// TIA Portal project "Centris" (V16)

(* hardware
DEVICE "S7-1200 station_1"  S7-1200 Station
   slot 0: "Rack_0"  S7-1200 Rack  Rack  V1.0
   slot 1: "PLC_1"  CPU 1214C DC/DC/Rly  6ES7 214-1HG40-0XB0  V4.4
*)

// ===== PLC "PLC_1"  CPU 1214C DC/DC/Rly =====

TYPE "UR__T2O_Robot"
   STRUCT
      "Controller major version" : USInt;
      "Controller minor version" : USInt;
      Reserved : UInt;
      "Robot mode" : USInt;
      "Real time machine seconds" : USInt;
      "Real time machine milliseconds" : UInt;
      "Real time machine minutes" : USInt;
      "Real time machine hours" : USInt;
      "Real time machine days" : UInt;
      "Robot current [A]" : Real;
      "PW: Is power on" : Bool;
      "PR: Is program running" : Bool;
      "TB: Is teach button pressed" : Bool;
      "PB: Is power button pressed" : Bool;
      Reserved_4 : Bool;
      Reserved_5 : Bool;
      Reserved_6 : Bool;
      Reserved_7 : Bool;
      Reserved_8_15 : USInt;
      Reserved_16_31 : UInt;
      "Speed slider fraction" : Real;
   END_STRUCT;
END_TYPE

TYPE "UR__T2O_Safety"
   STRUCT
      "Safety mode" : USInt;
      Reserved_1 : USInt;
      Reserved_2 : UInt;
      "NO: Is normal mode" : Bool;
      "RD: Is reduced mode" : Bool;
      "PS: Is protective stopped" : Bool;
      "RC: Is recovery mode" : Bool;
      "SS: Is safeguard stopped" : Bool;
      "SES: Is system emergency stopped" : Bool;
      "RES: Is robot emergency stopped" : Bool;
      "ES: Is emergency stopped" : Bool;
      "VL: Is violation" : Bool;
      "FT: Is fault" : Bool;
      "ST: Is stopped due to safety" : Bool;
      Reserved_11 : Bool;
      Reserved_12 : Bool;
      Reserved_13 : Bool;
      Reserved_14 : Bool;
      Reserved_15 : Bool;
      Reserved_16_31 : UInt;
   END_STRUCT;
END_TYPE

TYPE "UR__T2O_IOs"
   STRUCT
      "Standard digital inputs" : USInt;
      "Configurable digital inputs" : USInt;
      "Standard digital outputs" : USInt;
      "Configurable digital outputs" : USInt;
      "Analog I/O types" : USInt;
      Reserved_8_15 : USInt;
      Reserved_16_31 : UInt;
      "Standard analog input [A or V]" : Array[0..1] of Real;
      "Standard analog output [A or V]" : Array[0..1] of Real;
      "I/O current [A]" : Real;
      "Euromap67 input bits" : Array[0..31] of Bool;
      "Euromap67 output bits" : Array[0..31] of Bool;
      "Euromap67 24V voltage" : Real;
      "Euromap67 24V current" : Real;
   END_STRUCT;
END_TYPE

TYPE "UR__T2O_Tool"
   STRUCT
      "Tool mode" : USInt;
      Reserved_7_15 : USInt;
      Reserved_16_31 : UInt;
      "TDI: Tool Digital Inputs" : USInt;
      "TDO: Tool Digital Outputs" : USInt;
      "TAIT: Tool Analog Input Types" : USInt;
      Reserved_24_31 : USInt;
      "Tool analog input [A or V]" : Array[0..1] of Real;
      "Tool output voltage [V]" : Real;
      "Tool current [A]" : Real;
   END_STRUCT;
END_TYPE

TYPE "UR__O2T_floats"
   STRUCT
      Register : Array[0..11] of Real;
   END_STRUCT;
END_TYPE

TYPE "UR__O2T_ints"
   STRUCT
      Register : Array[0..11] of DInt;
   END_STRUCT;
END_TYPE

TYPE "UR__O2T_bits"
   STRUCT
      Register : Array[0..31] of Bool;
   END_STRUCT;
END_TYPE

TYPE "UR__O2T_Robot"
   STRUCT
      "SSM: Speed slider fraction mask" : Bool;
      Reserved_1 : Bool;
      Reserved_2 : Bool;
      Reserved_3 : Bool;
      Reserved_4 : Bool;
      Reserved_5 : Bool;
      Reserved_6 : Bool;
      Reserved_7 : Bool;
      Reserved_8_15 : USInt;
      Reserved_16_31 : UInt;
      "Speed slider fraction" : Real;
   END_STRUCT;
END_TYPE

TYPE "UR__O2T_IOs"
   STRUCT
      "Standard digital output mask" : USInt;
      "Configurable digital output mask" : USInt;
      "Standard digital outputs" : USInt;
      "Configurable digital outputs" : USInt;
      "AOM: Analog output mask" : USInt;
      "AOT: Analog output types" : USInt;
      "TDOM: Tool digital output mask" : USInt;
      "TDO: Tool digital output" : USInt;
      "Standard analog output" : Array[0..1] of Real;
   END_STRUCT;
END_TYPE

TYPE "Recipe_Data"
   STRUCT
      ID : DInt;   // ID
      ServoSpeed : DInt;
      ServoForceRamp : DInt;
      ServoForce : DInt;
      ServoRedPos : DInt;
      ServoBluePos : DInt;
      ServoYellowPos : DInt;
      "IV RedProgram" : Int;
      "IV BlueProgram" : Int;
      "IV YellowProgram" : Int;
   END_STRUCT;
END_TYPE

TYPE "Latch"
   STRUCT
      Latch : Bool;
      Ons : Bool;
      Action : Bool;
      Delay : Bool;
      PB : Bool;
      TON : IEC_TIMER;
   END_STRUCT;
END_TYPE

TYPE "UR_9_O2T_Registers"
   STRUCT
      Bits : "UR__O2T_bits";
      Ints : "UR__O2T_ints";
      Floats : "UR__O2T_floats";
   END_STRUCT;
END_TYPE

TYPE "UR_8_O2T_Robot_IO"
   STRUCT
      Robot : "UR__O2T_Robot";
      IOs : "UR__O2T_IOs";
   END_STRUCT;
END_TYPE

TYPE "UR_7_T2O_FloatRegisters"
   STRUCT
      Register : Array[0..23] of Real;
   END_STRUCT;
END_TYPE

TYPE "UR_6_T2O_IntRegisters"
   STRUCT
      Register : Array[0..23] of DInt;
   END_STRUCT;
END_TYPE

TYPE "UR_5_T2O_BitRegisters"
   STRUCT
      Register : Array[0..63] of Bool;
   END_STRUCT;
END_TYPE

TYPE "UR_4_T2O_TCP"
   STRUCT
      "TCP Position (X,Y,Z) [m]" : Array[0..2] of Real;
      "TCP Position (RX,RY,RZ) [rad]" : Array[0..2] of Real;
      "TCP velocity (X,Y,Z) [m/s]" : Array[0..2] of Real;
      "TCP velocity (RX,RY,RZ) [rad/s]" : Array[0..2] of Real;
      "TCP force (X,Y,Z) [N]" : Array[0..2] of Real;
      "TCP torque (X,Y,Z) [Nm]" : Array[0..2] of Real;
      "TCP force scalar [N]" : Real;
   END_STRUCT;
END_TYPE

TYPE "UR_3_T2O_Joints"
   STRUCT
      "Joint position [rad]" : Array[0..5] of Real;
      "Joint velocity [rad/s]" : Array[0..5] of Real;
      "Joint current [A]" : Array[0..5] of Real;
      "Joint temperature [°C]" : Array[0..5] of Real;
      "Joint mode" : Array[0..5] of USInt;
      Reserved_9 : UInt;
   END_STRUCT;
END_TYPE

TYPE "UR_2_T2O_IO"
   STRUCT
      IOs : "UR__T2O_IOs";
      Tool : "UR__T2O_Tool";
   END_STRUCT;
END_TYPE

TYPE "UR_1_T2O_State"
   STRUCT
      Robot : "UR__T2O_Robot";
      Safety : "UR__T2O_Safety";
   END_STRUCT;
END_TYPE

TYPE "Festo Control IN/OUT"
   STRUCT
      "Enable Connection" : Bool;
      "Device Type" : String;
      "Enable FPC" : Bool;
      "Enable FHPPPlus_In" : Int;
      "Enable FHPPPlus_Out" : Int;
      "IP_Oct#1" : Int;
      "IP_Oct#2" : Int;
      "IP_Oct#3" : Int;
      "IP_Oct#4" : Int;
      "Interface ID" : Hw_Any;
      "Connection ID" : Int;
      TimeOut : Time;
      "Com Enabled" : Bool;
      Error : Bool;
      Status : "DT_FML_STATUS";
      "Enable Control" : Bool;
      "Stop Control" : Bool;
      "Halt Control" : Bool;
      "Brake Control" : Bool;
      "Reset Control" : Bool;
      "HMI Access" : Bool;
      "Operation Mode" : Int;
      "Start Task" : Bool;
      "Start Homing" : Bool;
      "Jog Positive" : Bool;
      "Jog Negative" : Bool;
      "Teach Value" : Bool;
      "Clear Rem Position" : Bool;
      Relative : Bool;
      "Desactivate Stroke Limit" : Bool;
      "Execute Function" : Bool;
      "Record Number" : Int;
      "Set Function Number" : Int;
      "Set Function Group" : Int;
      "Set Velocity" : DInt;
      "Set Position Pre" : DInt;
      "Set Position Val" : DInt;
      "Set Force Ramp" : DInt;
      "Set Force" : DInt;
      "Set Rot Ramp" : DInt;
      "Set Rot Speed" : DInt;
      "Spare 1" : DInt;
      "Drive Enabled" : Bool;
      "Driver Ready" : Bool;
      Warning : Bool;
      "Driver Faulted" : Bool;
      "Driver Supply Voltage Present" : Bool;
      "Control FCT_HMI" : Bool;
      "Actual Operation Mode" : Int;
      "Halt Not Active" : Bool;
      "Start ACK" : Bool;
      "PLC Master Control" : Bool;
      "Teach ACK" : Bool;
      "Drive Moving" : Bool;
      "Drag Error" : Bool;
      "Stand Still Control" : Bool;
      "Homing Valid" : Bool;
      "Actual Record Number" : Int;
      RC1 : Bool;
      RCC : Bool;
      "Velocity Limit Reached" : Bool;
      "Stroke Limit Reached" : Bool;
      "Function Is Active" : Bool;
      "Actual Function Number" : Int;
      "Actual Function Group" : Int;
      "Actual Position" : DInt;
      "Actual Velocity" : DInt;
      "Actual Force" : DInt;
      "Actual Rot Ramp" : DInt;
      "Actual Rot Speed" : DInt;
      WatchDog_Timer_ON : Time;
      WatchDog_Timer_OFF : Time;
      WatrchDog_Reset : Bool;
      "Execute PNU" : Bool;
      Write : Bool;
      DatatypeWR : Int;
      PNU : Int;
      Subindex : Int;
      Value : DInt;
      Done : Bool;
      ErrorPNU : Bool;
      ActPNU : Int;
      ActSubindex : Int;
      ActValue : DInt;
      DatatypeRD : Int;
      StatusPNU : "DT_FML_STATUS";
      WatchDog_Timer : Array[0..10] of IEC_TIMER;
      WatchDog_Reset_Connection : Bool;
      WatchDog_Reset_Device : Bool;
      WatchDog_Reset_Control : Bool;
      "PNU BOOL" : Bool;
      "Manual Buffer" : DInt;
      "Position Buffer" : DInt;
      Delay : Array[0..10] of IEC_TIMER;
      SetProgram_Red : Int;
      SetProgram_Blue : Int;
      SetProgram_Yellow : Int;
      Set_Red_Position : DInt;
      Set_Blue_Position : DInt;
      Set_Yellow_Position : DInt;
      Red_StartTask : Bool;
      Blue_StartTask : Bool;
      Yellow_StartTask : Bool;
      Home_StartTask : Bool;
      RedPos : Bool;
      BluePos : Bool;
      YellowPos : Bool;
      HomePos : Bool;
      Available_StartTask : Bool;
   END_STRUCT;
END_TYPE

TYPE "Safety"
   STRUCT
      "EStops OK" : Bool;
      "Safety Guards OK" : Bool;
      "Interlocks OK" : Bool;
      "SSD Robots OK" : Bool;
      "SSD Servos OK" : Bool;
      "Safety Doors OK" : Bool;
      "Safety Relays OK" : Bool;
      "SSD vfd Motors OK" : Bool;
      "Safety Curtains OK" : Bool;
      "Safety Devices OK" : Bool;
      "Communication Devices OK" : Bool;
      "Clear Error Devices OK" : Bool;
      "Clear Fault Devices OK" : Bool;
      "Safety Air OK" : Bool;
      "Power ON Start" : Bool;
      "Enable System Start" : Bool;
      "All Safety Devices OK" : Bool;
   END_STRUCT;
END_TYPE

TYPE "Mode"
   STRUCT
      "Run Stop" : Bool;
      "Run Auto" : Bool;
      "Run Start" : Bool;
      "Run Manual" : Bool;
      "Run Dry Cycle" : Bool;
      "Enable Cycle Stop" : Bool;
      "Enable Auto" : Bool;
      "Enable Start" : Bool;
      "Enable Manual" : Bool;
      "Enable Dry Cycle" : Bool;
      "Enable Home" : Bool;
      "Run Home" : Bool;
   END_STRUCT;
END_TYPE

TYPE "Push_Buttons"
   STRUCT
      AllHome : Bool;
      Stop : Bool;
      Auto : Bool;
      Start : Bool;
      StartProcess : Bool;
      Manual : Bool;
      DryCycle : Bool;
      Reset : Bool;
      Trigger : Bool;
      IVProgramRed : Bool;
      IVProgramBLue : Bool;
      IVProgramYellow : Bool;
      FestoRedPos : Bool;
      FestoBluePos : Bool;
      FestoYellowPos : Bool;
      FestoHomePos : Bool;
      "UR RedPos" : Bool;
      "UR BluePos" : Bool;
      "UR YellowPos" : Bool;
      "UR HomePos" : Bool;
      RecipeSelect : Array[0..5] of Bool;
      RecipeEdit : Array[0..5] of Bool;
      Saving : Bool;
      ResetBuffer : Bool;
      AutoPlay : Bool;
      AutoInit : Bool;
      StartProgram : Bool;
      StopProgram : Bool;
      PauseProgram : Bool;
      FreeDrive : Bool;
      FestoReset : Bool;
      URReset : Bool;
      MainReset : Bool;
      VisionReset : Bool;
      FaultsReset : Bool;
      WarningsReset : Bool;
   END_STRUCT;
END_TYPE

TYPE "UR_O2T"
   STRUCT
      "Robot IO" : "UR_8_O2T_Robot_IO";
      "Reg 1" : "UR_9_O2T_Registers";
      "Reg 2" : "UR_9_O2T_Registers";
   END_STRUCT;
END_TYPE

TYPE "Alarms"
   STRUCT
      Fault : Array[0..100] of Bool;
      Warning : Array[0..100] of Bool;
      Status : Array[0..100] of Bool;
      Clear : Array[0..100] of Bool;
      ClearFaults : Bool;
      ClearWarnings : Bool;
      ClearStatus : Bool;
      Fton : Array[0..100] of IEC_TIMER;
      Wton : Array[0..100] of IEC_TIMER;
      Ston : Array[0..100] of IEC_TIMER;
   END_STRUCT;
END_TYPE

TYPE "Ctlr_Recipe"
   STRUCT
      "Actual Running Recipe" : "Recipe_Data";
      "Editing Recipe" : "Recipe_Data";
      "Selected Recipe" : "Recipe_Data";
      Saving : "Latch";
      Select : "Latch";
      Edit : "Latch";
      MoveBit : Array[0..5] of Bool;
      EditBit : Array[0..5] of Bool;
      "Any Recipe Selected" : Bool;
      "None Recipe Selected" : Bool;
      "End Of Sequence" : Bool;
      "Cycle Running" : Bool;
   END_STRUCT;
END_TYPE

TYPE "iv_500ca_in"
   STRUCT
      "Trigger response" : Bool;   // Command Status Bits Address 0:0
      "Master registration response" : Bool;   // Command Status Bits Address 0:1
      "Program switching response" : Bool;   // Command Status Bits Address 0:2
      "Warning clear response" : Bool;   // Command Status Bits Address 0:3
      "Statistics reset response" : Bool;   // Command Status Bits Address 0:4
      "Buffer clear response" : Bool;   // Command Status Bits Address 0:5
      "Command Status Bits Address 0:6" : Bool;   // Command Status Bits Address 0:6
      "Command Status Bits Address 0:7" : Bool;   // Command Status Bits Address 0:7
      "Trigger failed" : Bool;   // Command Status Bits Address 1:0
      "Master registration failed" : Bool;   // Command Status Bits Address 1:1
      "Program switching failed" : Bool;   // Command Status Bits Address 1:2
      "Command Status Bits Address 1:3" : Bool;   // Command Status Bits Address 1:3
      "Command Status Bits Address 1:4" : Bool;   // Command Status Bits Address 1:4
      "Command Status Bits Address 1:5" : Bool;   // Command Status Bits Address 1:5
      "Command Status Bits Address 1:6" : Bool;   // Command Status Bits Address 1:6
      "Command Status Bits Address 1:7" : Bool;   // Command Status Bits Address 1:7
      "Result available" : Bool;   // Command Status Bits Address 2:0
      "Result update complete" : Bool;   // Command Status Bits Address 2:1
      Busy : Bool;   // Command Status Bits Address 2:2
      Imaging : Bool;   // Command Status Bits Address 2:3
      RUN : Bool;   // Command Status Bits Address 2:4
      Ready : Bool;   // Command Status Bits Address 2:5
      "Command Status Bits Address 2:6" : Bool;   // Command Status Bits Address 2:6
      "Command Status Bits Address 2:7" : Bool;   // Command Status Bits Address 2:7
      "Command Status Bits Address 3:0" : Bool;   // Command Status Bits Address 3:0
      "Command Status Bits Address 3:1" : Bool;   // Command Status Bits Address 3:1
      "Command Status Bits Address 3:2" : Bool;   // Command Status Bits Address 3:2
      "Command Status Bits Address 3:3" : Bool;   // Command Status Bits Address 3:3
      "Command Status Bits Address 3:4" : Bool;   // Command Status Bits Address 3:4
      "Buffer overrun status" : Bool;   // Command Status Bits Address 3:5
      "Warning status" : Bool;   // Command Status Bits Address 3:6
      "Error status" : Bool;   // Command Status Bits Address 3:7
      "Overall judgment" : Bool;   // Device Results Bits Address 0:0
      "Position correction" : Bool;   // Device Results Bits Address 0:1
      "Logic 1" : Bool;   // Device Results Bits Address 0:2
      "Logic 2" : Bool;   // Device Results Bits Address 0:3
      "Logic 3" : Bool;   // Device Results Bits Address 0:4
      "Logic 4" : Bool;   // Device Results Bits Address 0:5
      "Overall judgement NG" : Bool;   // Device Results Bits Address 0:6
      "Device Results Bits Address 0:7" : Bool;   // Device Results Bits Address 0:7
      "Device Results Bits Address 1:0" : Bool;   // Device Results Bits Address 1:0
      "Device Results Bits Address 1:1" : Bool;   // Device Results Bits Address 1:1
      "Device Results Bits Address 1:2" : Bool;   // Device Results Bits Address 1:2
      "Device Results Bits Address 1:3" : Bool;   // Device Results Bits Address 1:3
      "Device Results Bits Address 1:4" : Bool;   // Device Results Bits Address 1:4
      "Device Results Bits Address 1:5" : Bool;   // Device Results Bits Address 1:5
      "Device Results Bits Address 1:6" : Bool;   // Device Results Bits Address 1:6
      "Device Results Bits Address 1:7" : Bool;   // Device Results Bits Address 1:7
      "Tool 1" : Bool;   // Device Results Bits Address 2:0
      "Tool 2" : Bool;   // Device Results Bits Address 2:1
      "Tool 3" : Bool;   // Device Results Bits Address 2:2
      "Tool 4" : Bool;   // Device Results Bits Address 2:3
      "Tool 5" : Bool;   // Device Results Bits Address 2:4
      "Tool 6" : Bool;   // Device Results Bits Address 2:5
      "Tool 7" : Bool;   // Device Results Bits Address 2:6
      "Tool 8" : Bool;   // Device Results Bits Address 2:7
      "Tool 9" : Bool;   // Device Results Bits Address 3:0
      "Tool 10" : Bool;   // Device Results Bits Address 3:1
      "Tool 11" : Bool;   // Device Results Bits Address 3:2
      "Tool 12" : Bool;   // Device Results Bits Address 3:3
      "Tool 13" : Bool;   // Device Results Bits Address 3:4
      "Tool 14" : Bool;   // Device Results Bits Address 3:5
      "Tool 15" : Bool;   // Device Results Bits Address 3:6
      "Tool 16" : Bool;   // Device Results Bits Address 3:7
      "Error code" : Word;   // Device Status Words Address 0 to 1
      "Warning code" : Word;   // Device Status Words Address 2 to 3
      "Number of remaining buffers" : Word;   // Device Status Words Address 4 to 5
      Checksum : Word;   // Device Status Words Address 6 to 7
      "Current program No." : Word;   // Device Status Words Address 8 to 9
      "Program No. during judgment" : Word;   // Device Status Words Address 10 to 11
      "Result No." : Word;   // Device Status Words Address 12 to 13
      "Processing time" : Word;   // Device Status Words Address 14 to 15
      "Processing time Max" : Word;   // Device Statistics Address 0 to 1
      "Processing time Min" : Word;   // Device Statistics Address 2 to 3
      "Processing time Ave" : Word;   // Device Statistics Address 4 to 5
      "Device Statistics Address 6 to 7" : Word;   // Device Statistics Address 6 to 7
      "Number of triggers" : DWord;   // Device Statistics Address 8 to 11
      "Number of OKs" : DWord;   // Device Statistics Address 12 to 15
      "Number of NGs" : DWord;   // Device Statistics Address 16 to 19
      "Number of trigger errors" : DWord;   // Device Statistics Address 20 to 23
      "Device Statistics Address 24 to 27" : DWord;   // Device Statistics Address 24 to 27
      "Position correction tool matching rate" : Word;   // Position Adjust Result Address 0 to 1
      "Position correction score MAX" : Word;   // Position Adjust Result Address 2 to 3
      "Position correction score MIN" : Word;   // Position Adjust Result Address 4 to 5
      "Position correction tool Threshold value" : Word;   // Position Adjust Result Address 6 to 7
      "Position Adjust Result Address 8 to 9" : Word;   // Position Adjust Result Address 8 to 9
      "Position Adjust Result Address 10 to 11" : Word;   // Position Adjust Result Address 10 to 11
      "Position Adjust Result Address 12 to 13" : Word;   // Position Adjust Result Address 12 to 13
      "Position Adjust Result Address 14 to 15" : Word;   // Position Adjust Result Address 14 to 15
      "Position Adjust Result Address 16 to 17" : Word;   // Position Adjust Result Address 16 to 17
      "Position Adjust Result Address 18 to 19" : Word;   // Position Adjust Result Address 18 to 19
      "Tool 1 matching rate" : Word;   // Tool Result Address 0 to 1
      "Tool 1 matching rate MAX" : Word;   // Tool Result Address 2 to 3
      "Tool 1 matching rate MIN" : Word;   // Tool Result Address 4 to 5
      "Tool 1 lower limit value" : Word;   // Tool Result Address 6 to 7
      "Tool 1 upper limit value" : Word;   // Tool Result Address 8 to 9
      "Tool Result Address 10" : Byte;   // Tool Result Address 10
      "Tool Result Address 11" : Byte;   // Tool Result Address 11
      "Tool Result Address 12" : Byte;   // Tool Result Address 12
      "Tool Result Address 13" : Byte;   // Tool Result Address 13
      "Tool Result Address 14" : Byte;   // Tool Result Address 14
      "Tool Result Address 15" : Byte;   // Tool Result Address 15
      "Tool Result Address 16" : Byte;   // Tool Result Address 16
      "Tool Result Address 17" : Byte;   // Tool Result Address 17
      "Tool Result Address 18" : Byte;   // Tool Result Address 18
      "Tool Result Address 19" : Byte;   // Tool Result Address 19
   END_STRUCT;
END_TYPE

TYPE "iv_500ca_out"
   STRUCT
      "Trigger request" : Bool;   // Command Control 1:0
      "Master registration request" : Bool;   // Command Control 1:1
      "Programm switching request" : Bool;   // Command Control 1:2
      "Warning clear request" : Bool;   // Command Control 1:3
      "Statistics reset request" : Bool;   // Command Control 1:4
      "Buffer clear request" : Bool;   // Command Control 1:5
      "Command Control 1:6" : Bool;   // Command Control 1:6
      "Command Control 1:7" : Bool;   // Command Control 1:7
      "Result acquisition complete notification" : Bool;   // Command Control 2:0
      "Command Control 2:1" : Bool;   // Command Control 2:1
      "Command Control 2:2" : Bool;   // Command Control 2:2
      "Command Control 2:3" : Bool;   // Command Control 2:3
      "Command Control 2:4" : Bool;   // Command Control 2:4
      "Command Control 2:5" : Bool;   // Command Control 2:5
      "Command Control 2:6" : Bool;   // Command Control 2:6
      "Command Control 2:7" : Bool;   // Command Control 2:7
      "Command Control 3" : Byte;   // Command Control 3
      "Programm No." : Word;   // Command Control 4 to 5
      "Command Control 6" : Byte;   // Command Control 6
      "Command Control 7" : Byte;   // Command Control 7
      "Command Control 8" : Byte;   // Command Control 8
      "Command Control 9" : Byte;   // Command Control 9
      "Command Control 10" : Byte;   // Command Control 10
      "Command Control 11" : Byte;   // Command Control 11
   END_STRUCT;
END_TYPE

TYPE "IV_Ctrl"
   STRUCT
      CommActive : Bool;
      ResetBuffer : Bool;
      InspectionComplete : Bool;
      InspectionOK : Bool;
      InspectionNOK : Bool;
      InspectionRequest : Bool;
      InspectReqTimeout : IEC_TIMER;
      ConnectionFault : Bool;
      CameraFault : Bool;
      InspectionRequestTimeoutFault : Bool;
      "Clear Results" : Bool;
      Trigger : Bool;
      OKRed : Bool;
      NOKRed : Bool;
      OKBlue : Bool;
      NOKBlue : Bool;
      OKYellow : Bool;
      NOKYellow : Bool;
      AllClearResults : Bool;
      NOKAllResults : Bool;
      "Run Red" : Bool;
      "Run Blue" : Bool;
      "Run Yellow" : Bool;
      OKAnyResult : Bool;
   END_STRUCT;
END_TYPE

TYPE "PLC_Digital_IN"
   STRUCT
      START : Bool;
      RESET : Bool;
      ESTOP : Bool;
      "I0.3" : Bool;
      "I0.4" : Bool;
      "I0.5" : Bool;
      "I0.6" : Bool;
      "I0.7" : Bool;
      "I1.0" : Bool;
      "I1.1" : Bool;
      "I1.2" : Bool;
      "I1.3" : Bool;
      "I1.4" : Bool;
      "I1.5" : Bool;
      "I1.6" : Bool;
      "I1.7" : Bool;
   END_STRUCT;
END_TYPE

TYPE "PLC_Digital_Out"
   STRUCT
      "Q0.0" : Bool;
      "Q0.1" : Bool;
      "Q0.2" : Bool;
      "Q0.3" : Bool;
      "Q0.4" : Bool;
      "Q0.5" : Bool;
      "Q0.6" : Bool;
      "Q0.7" : Bool;
      "Q1.0" : Bool;
      "Q1.1" : Bool;
      "Q1.2" : Bool;
      "Q1.3" : Bool;
      "Q1.4" : Bool;
      "Q1.5" : Bool;
      "Q1.6" : Bool;
      "Q1.7" : Bool;
   END_STRUCT;
END_TYPE

TYPE "UR_T2O"
   STRUCT
      State : "UR_1_T2O_State";
      IO : "UR_2_T2O_IO";
      Joints : "UR_3_T2O_Joints";
      TCP : "UR_4_T2O_TCP";
      Bits : "UR_5_T2O_BitRegisters";
      Ints : "UR_6_T2O_IntRegisters";
      Floats : "UR_7_T2O_FloatRegisters";
   END_STRUCT;
END_TYPE

TYPE "Production"
   STRUCT
      Ton : Array[0..12] of IEC_TIMER;
      Seq : Array[0..12] of Bool;
      Permissive : Array[0..12] of Bool;
      Clear : Array[0..12] of Bool;
      "Clear Sequence" : Bool;
      "All Home OK" : Bool;
      ReplaceIN : Array[0..15] of Bool;
      "Cycle ResetAllMemories" : Bool;
      "UR Home OK" : Bool;
      "UR Program" : DInt;
      "UR EndRoutine" : Bool;
      "All Memories StatusClear" : Bool;
      StatusSeq : Bool;
      StatusStart : Bool;
      StatusHome : Bool;
      "UR RunRed" : Bool;
      "UR RunBlue" : Bool;
      "UR RunYellow" : Bool;
      "UR Start Program" : Bool;
   END_STRUCT;
END_TYPE

// folder: FML DATATYPES

TYPE "DT_FML_STATUS"
   STRUCT
      Err : Bool;
      Cat : Int;
      ID : DInt;
   END_STRUCT;
END_TYPE

TYPE "DT_FML_PRM_FILE"
   STRUCT
      Control : Int;
      BitSequenceNr : Int;
      Data : Array[1..6] of Byte;
   END_STRUCT;
END_TYPE

TYPE "DT_FML_REF"
   STRUCT
      InData : Struct
         FHPP : Array[1..16] of Byte;
         FPC : Array[1..8] of Byte;
         FHPPplus : Array[1..10] of DInt;
      END_STRUCT;
      OutData : Struct
         FHPP : Array[1..16] of Byte;
         FPC : Array[1..8] of Byte;
         FHPPplus : Array[1..10] of DInt;
      END_STRUCT;
      Modbus : Bool;
      DeviceType : String[16];
      MemberID : Int;
      MemberIDmax : Int;
      Done : Bool;
      Err : Bool;
      PNU : Word;
      ActPNU : Word;
      ReqID : Int;
      RespID : Int;
      FPCC_Modus : Byte;
      FPCS_Modus : Byte;
      FPCC_Packet : "DT_FML_PRM_FILE";
      FPCS_Packet : "DT_FML_PRM_FILE";
      Subindex : Byte;
      ActSubindex : Byte;
      DatatypeWR : Byte;
      DatatypeRD : Byte;
      ParamValueWR : DInt;
      ParamValueRD : DInt;
   END_STRUCT;
END_TYPE

TYPE "DT_MB_CLIENT_INPUT"
   STRUCT
      REQ : Bool;
      DISCONNECT : Bool;
      Done : Bool;
      Busy : Bool;
      Error : Bool;
      MB_MODE : USInt;
      MB_DATA_ADDR : UDInt;
      MB_DATA_LEN : UInt;
   END_STRUCT;
END_TYPE

TYPE "DT_FML_PRM_DESCRIPTION"
   STRUCT
      PNU : Word;
      SUBINDEX : Byte;
      ACCESS : Byte;
      VALUE : DInt;
      LENGTH : Byte;
   END_STRUCT;
END_TYPE

TYPE "DT_FML_PRM_DIAGMESSAGE"
   STRUCT
      Event : DInt;
      MsgNumber : DInt;
      TimeStamp : DWord;
   END_STRUCT;
END_TYPE

// folder: (top level)

DATA_BLOCK "DB"   // DB1
{ S7_Optimized_Access := 'FALSE' }
VERSION : 0.1
   VAR
      Alarm : "Alarms";
      Prod : "Production";
      UR : "Production";
      Ctrl_Recipe : "Ctlr_Recipe";
      FESTO : "Festo Control IN/OUT";
      AUTO : "Festo Control IN/OUT";
      MANUAL : "Festo Control IN/OUT";
      OP : "Festo Control IN/OUT";
      HMI : "Push_Buttons";
      "Mod" : "Mode";
      Safe : "Safety";
      "IV Ctrl" : "IV_Ctrl";
      I : "PLC_Digital_IN";
      "N/A" : Bool;
   END_VAR
BEGIN
END_DATA_BLOCK

DATA_BLOCK "FHPP_MB_CLIENT_DB"   // DB7
{ S7_Optimized_Access := 'TRUE' }
AUTHOR : FESTO
FAMILY : E-DRIVE
VERSION : 5.1
// stored: InstanceOfName FHPP_MB_CLIENT
"FHPP_MB_CLIENT"
BEGIN
END_DATA_BLOCK

DATA_BLOCK "FHPP_CTRL_DB"   // DB8
{ S7_Optimized_Access := 'TRUE' }
AUTHOR : FESTO
FAMILY : E-DRIVE
VERSION : 5.1
// stored: InstanceOfName FHPP_CTRL
"FHPP_CTRL"
BEGIN
END_DATA_BLOCK

DATA_BLOCK "FPC_PNU_DB"   // DB9
{ S7_Optimized_Access := 'TRUE' }
AUTHOR : FESTO
FAMILY : E-DRIVE
VERSION : 5.1
// stored: InstanceOfName FPC_PNU
"FPC_PNU"
BEGIN
END_DATA_BLOCK

// folder: RECIPE

DATA_BLOCK "Recipe"   // DB2
{ S7_Optimized_Access := 'TRUE' }
VERSION : 0.1
BEGIN
END_DATA_BLOCK

// folder: UTILITIES OR DEVICES/FESTO

DATA_BLOCK "Global_Modbuss_CMMO"   // DB6
{ S7_Optimized_Access := 'TRUE' }
VERSION : 0.1
   VAR
      CMMO_REF : "DT_FML_REF";
   END_VAR
BEGIN
END_DATA_BLOCK

DATA_BLOCK "gBUFFER_MODBUS"   // DB100
TITLE = Buffer for MB_Client
{ S7_Optimized_Access := 'FALSE' }
AUTHOR : FESTO
FAMILY : E-Drives
VERSION : 4.1
   VAR
      ModbusBuffer : Array[1..100] of Byte;
   END_VAR
BEGIN
END_DATA_BLOCK

// folder: UTILITIES OR DEVICES/MODBUS TCP LABVIEW

DATA_BLOCK "Labview"   // DB3
{ S7_Optimized_Access := 'FALSE' }
VERSION : 0.1
BEGIN
END_DATA_BLOCK

DATA_BLOCK "MBConfig"   // DB4
{ S7_Optimized_Access := 'FALSE' }
VERSION : 0.1
BEGIN
END_DATA_BLOCK

DATA_BLOCK "MBData"   // DB5
{ S7_Optimized_Access := 'FALSE' }
VERSION : 0.1
BEGIN
END_DATA_BLOCK

// folder: (top level)

ORGANIZATION_BLOCK "Main"   // OB1, LAD, ProgramCycle
TITLE = "Main Program Sweep (Cycle)"
{ S7_Optimized_Access := 'TRUE' }
VERSION : 0.1
   VAR_INPUT
      Initial_Call : Bool;   // Initial call of this OB
      Remanence : Bool;   // =True, if remanent data are available
   END_VAR
BEGIN

REGION Network 1: CALL_LADDER
END_REGION

REGION Network 2: FESTO MODBUS CLIENT
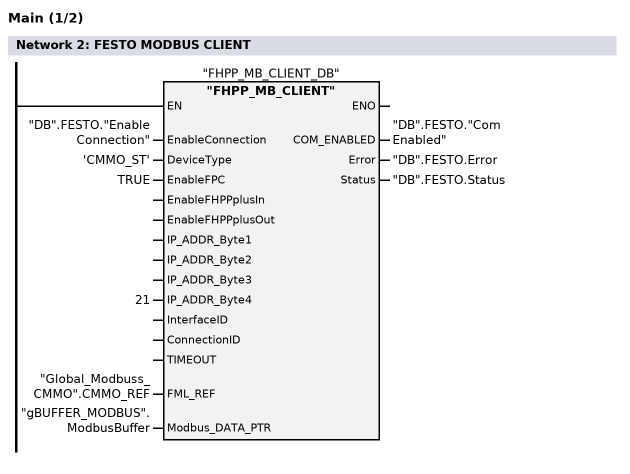
   RUNG wire#powerrail
      "FHPP_MB_CLIENT_DB"(EnableConnection := "DB".FESTO."Enable Connection", DeviceType := 'CMMO_ST', EnableFPC := TRUE, EnableFHPPplusIn :=, EnableFHPPplusOut :=, IP_ADDR_Byte1 :=, IP_ADDR_Byte2 :=, IP_ADDR_Byte3 :=, IP_ADDR_Byte4 := 21, InterfaceID :=, ConnectionID :=, TIMEOUT :=, FML_REF := "Global_Modbuss_CMMO".CMMO_REF, Modbus_DATA_PTR := "gBUFFER_MODBUS".ModbusBuffer, COM_ENABLED => "DB".FESTO."Com Enabled", Error => "DB".FESTO.Error, Status => "DB".FESTO.Status)
   END_RUNG
   // the same network as SCL:
   "FHPP_MB_CLIENT_DB"(EnableConnection := "DB".FESTO."Enable Connection",   // "FHPP_MB_CLIENT"
                       DeviceType := 'CMMO_ST',
                       EnableFPC := TRUE,
                       IP_ADDR_Byte4 := 21,
                       FML_REF := "Global_Modbuss_CMMO".CMMO_REF,
                       Modbus_DATA_PTR := "gBUFFER_MODBUS".ModbusBuffer,
                       COM_ENABLED => "DB".FESTO."Com Enabled",
                       Error => "DB".FESTO.Error,
                       Status => "DB".FESTO.Status);
END_REGION

REGION Network 3: FESTO DRIVER CONTROL
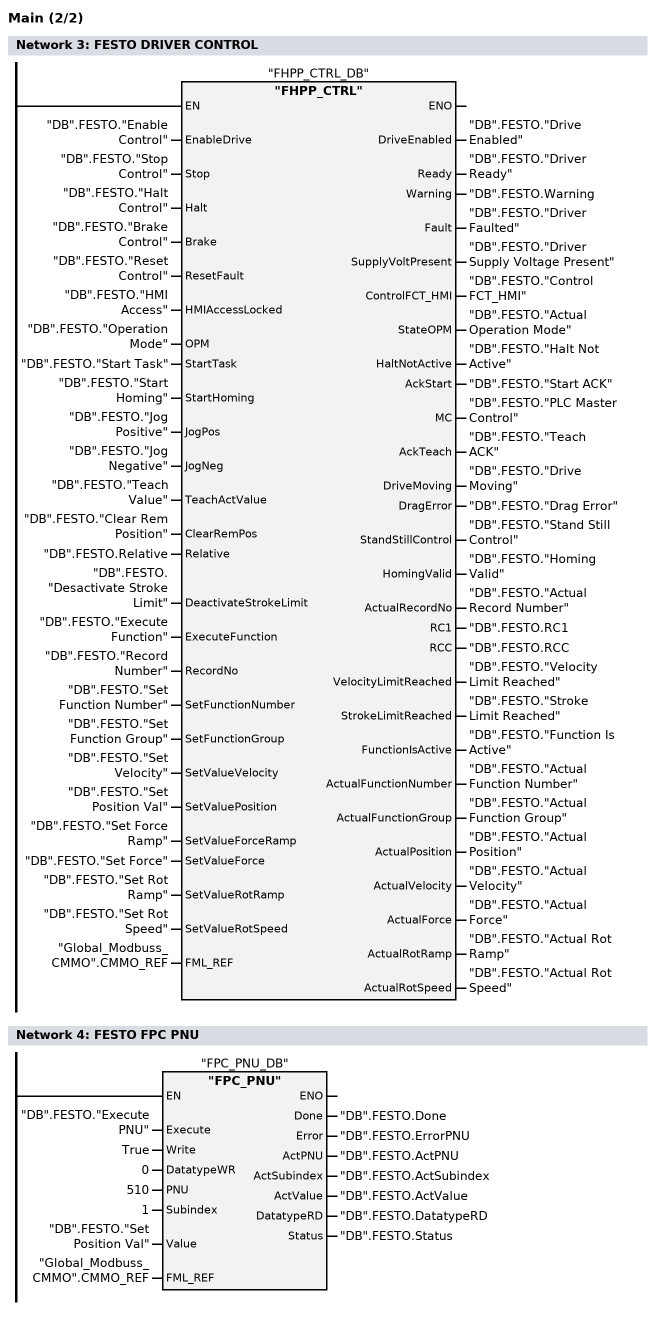
   RUNG wire#powerrail
      "FHPP_CTRL_DB"(EnableDrive := "DB".FESTO."Enable Control", Stop := "DB".FESTO."Stop Control", Halt := "DB".FESTO."Halt Control", Brake := "DB".FESTO."Brake Control", ResetFault := "DB".FESTO."Reset Control", HMIAccessLocked := "DB".FESTO."HMI Access", OPM := "DB".FESTO."Operation Mode", StartTask := "DB".FESTO."Start Task", StartHoming := "DB".FESTO."Start Homing", JogPos := "DB".FESTO."Jog Positive", JogNeg := "DB".FESTO."Jog Negative", TeachActValue := "DB".FESTO."Teach Value", ClearRemPos := "DB".FESTO."Clear Rem Position", Relative := "DB".FESTO.Relative, DeactivateStrokeLimit := "DB".FESTO."Desactivate Stroke Limit", ExecuteFunction := "DB".FESTO."Execute Function", RecordNo := "DB".FESTO."Record Number", SetFunctionNumber := "DB".FESTO."Set Function Number", SetFunctionGroup := "DB".FESTO."Set Function Group", SetValueVelocity := "DB".FESTO."Set Velocity", SetValuePosition := "DB".FESTO."Set Position Val", SetValueForceRamp := "DB".FESTO."Set Force Ramp", SetValueForce := "DB".FESTO."Set Force", SetValueRotRamp := "DB".FESTO."Set Rot Ramp", SetValueRotSpeed := "DB".FESTO."Set Rot Speed", FML_REF := "Global_Modbuss_CMMO".CMMO_REF, DriveEnabled => "DB".FESTO."Drive Enabled", Ready => "DB".FESTO."Driver Ready", Warning => "DB".FESTO.Warning, Fault => "DB".FESTO."Driver Faulted", SupplyVoltPresent => "DB".FESTO."Driver Supply Voltage Present", ControlFCT_HMI => "DB".FESTO."Control FCT_HMI", StateOPM => "DB".FESTO."Actual Operation Mode", HaltNotActive => "DB".FESTO."Halt Not Active", AckStart => "DB".FESTO."Start ACK", MC => "DB".FESTO."PLC Master Control", AckTeach => "DB".FESTO."Teach ACK", DriveMoving => "DB".FESTO."Drive Moving", DragError => "DB".FESTO."Drag Error", StandStillControl => "DB".FESTO."Stand Still Control", HomingValid => "DB".FESTO."Homing Valid", ActualRecordNo => "DB".FESTO."Actual Record Number", RC1 => "DB".FESTO.RC1, RCC => "DB".FESTO.RCC, VelocityLimitReached => "DB".FESTO."Velocity Limit Reached", StrokeLimitReached => "DB".FESTO."Stroke Limit Reached", FunctionIsActive => "DB".FESTO."Function Is Active", ActualFunctionNumber => "DB".FESTO."Actual Function Number", ActualFunctionGroup => "DB".FESTO."Actual Function Group", ActualPosition => "DB".FESTO."Actual Position", ActualVelocity => "DB".FESTO."Actual Velocity", ActualForce => "DB".FESTO."Actual Force", ActualRotRamp => "DB".FESTO."Actual Rot Ramp", ActualRotSpeed => "DB".FESTO."Actual Rot Speed")
   END_RUNG
   // the same network as SCL:
   "FHPP_CTRL_DB"(EnableDrive := "DB".FESTO."Enable Control",   // "FHPP_CTRL"
                  Stop := "DB".FESTO."Stop Control",
                  Halt := "DB".FESTO."Halt Control",
                  Brake := "DB".FESTO."Brake Control",
                  ResetFault := "DB".FESTO."Reset Control",
                  HMIAccessLocked := "DB".FESTO."HMI Access",
                  OPM := "DB".FESTO."Operation Mode",
                  StartTask := "DB".FESTO."Start Task",
                  StartHoming := "DB".FESTO."Start Homing",
                  JogPos := "DB".FESTO."Jog Positive",
                  JogNeg := "DB".FESTO."Jog Negative",
                  TeachActValue := "DB".FESTO."Teach Value",
                  ClearRemPos := "DB".FESTO."Clear Rem Position",
                  Relative := "DB".FESTO.Relative,
                  DeactivateStrokeLimit := "DB".FESTO."Desactivate Stroke Limit",
                  ExecuteFunction := "DB".FESTO."Execute Function",
                  RecordNo := "DB".FESTO."Record Number",
                  SetFunctionNumber := "DB".FESTO."Set Function Number",
                  SetFunctionGroup := "DB".FESTO."Set Function Group",
                  SetValueVelocity := "DB".FESTO."Set Velocity",
                  SetValuePosition := "DB".FESTO."Set Position Val",
                  SetValueForceRamp := "DB".FESTO."Set Force Ramp",
                  SetValueForce := "DB".FESTO."Set Force",
                  SetValueRotRamp := "DB".FESTO."Set Rot Ramp",
                  SetValueRotSpeed := "DB".FESTO."Set Rot Speed",
                  FML_REF := "Global_Modbuss_CMMO".CMMO_REF,
                  DriveEnabled => "DB".FESTO."Drive Enabled",
                  Ready => "DB".FESTO."Driver Ready",
                  Warning => "DB".FESTO.Warning,
                  Fault => "DB".FESTO."Driver Faulted",
                  SupplyVoltPresent => "DB".FESTO."Driver Supply Voltage Present",
                  ControlFCT_HMI => "DB".FESTO."Control FCT_HMI",
                  StateOPM => "DB".FESTO."Actual Operation Mode",
                  HaltNotActive => "DB".FESTO."Halt Not Active",
                  AckStart => "DB".FESTO."Start ACK",
                  MC => "DB".FESTO."PLC Master Control",
                  AckTeach => "DB".FESTO."Teach ACK",
                  DriveMoving => "DB".FESTO."Drive Moving",
                  DragError => "DB".FESTO."Drag Error",
                  StandStillControl => "DB".FESTO."Stand Still Control",
                  HomingValid => "DB".FESTO."Homing Valid",
                  ActualRecordNo => "DB".FESTO."Actual Record Number",
                  RC1 => "DB".FESTO.RC1,
                  RCC => "DB".FESTO.RCC,
                  VelocityLimitReached => "DB".FESTO."Velocity Limit Reached",
                  StrokeLimitReached => "DB".FESTO."Stroke Limit Reached",
                  FunctionIsActive => "DB".FESTO."Function Is Active",
                  ActualFunctionNumber => "DB".FESTO."Actual Function Number",
                  ActualFunctionGroup => "DB".FESTO."Actual Function Group",
                  ActualPosition => "DB".FESTO."Actual Position",
                  ActualVelocity => "DB".FESTO."Actual Velocity",
                  ActualForce => "DB".FESTO."Actual Force",
                  ActualRotRamp => "DB".FESTO."Actual Rot Ramp",
                  ActualRotSpeed => "DB".FESTO."Actual Rot Speed");
END_REGION

REGION Network 4: FESTO FPC PNU
   RUNG wire#powerrail
      "FPC_PNU_DB"(Execute := "DB".FESTO."Execute PNU", Write := True, DatatypeWR := 0, PNU := 510, Subindex := 1, Value := "DB".FESTO."Set Position Val", FML_REF := "Global_Modbuss_CMMO".CMMO_REF, Done => "DB".FESTO.Done, Error => "DB".FESTO.ErrorPNU, ActPNU => "DB".FESTO.ActPNU, ActSubindex => "DB".FESTO.ActSubindex, ActValue => "DB".FESTO.ActValue, DatatypeRD => "DB".FESTO.DatatypeRD, Status => "DB".FESTO.Status)
   END_RUNG
   // the same network as SCL:
   "FPC_PNU_DB"(Execute := "DB".FESTO."Execute PNU",   // "FPC_PNU"
                Write := True,
                DatatypeWR := 0,
                PNU := 510,
                Subindex := 1,
                Value := "DB".FESTO."Set Position Val",
                FML_REF := "Global_Modbuss_CMMO".CMMO_REF,
                Done => "DB".FESTO.Done,
                Error => "DB".FESTO.ErrorPNU,
                ActPNU => "DB".FESTO.ActPNU,
                ActSubindex => "DB".FESTO.ActSubindex,
                ActValue => "DB".FESTO.ActValue,
                DatatypeRD => "DB".FESTO.DatatypeRD,
                Status => "DB".FESTO.Status);
END_REGION

REGION Network 5: LABVIEW MODBUS CLIENT
END_REGION

REGION Network 6: LABVIEW RESULT
END_REGION
END_ORGANIZATION_BLOCK

// folder: ALARMS

FUNCTION "FAULTS" : Void   // FC1, LAD
{ S7_Optimized_Access := 'TRUE' }
VERSION : 0.1
BEGIN
END_FUNCTION

FUNCTION "WARNINGS" : Void   // FC3, LAD
{ S7_Optimized_Access := 'TRUE' }
VERSION : 0.1
BEGIN
END_FUNCTION

FUNCTION "STATUS_MACHINE" : Void   // FC4, LAD
{ S7_Optimized_Access := 'TRUE' }
VERSION : 0.1
BEGIN
END_FUNCTION

// folder: HOME

FUNCTION "HOME" : Void   // FC2, LAD
{ S7_Optimized_Access := 'TRUE' }
VERSION : 0.1
BEGIN
END_FUNCTION

// folder: RECIPE

FUNCTION "SET RUN SELECT RECIPE" : Void   // FC11, LAD
{ S7_Optimized_Access := 'TRUE' }
VERSION : 0.1
BEGIN
END_FUNCTION

FUNCTION "SET VALUES FROM RECIPE" : Void   // FC13, LAD
{ S7_Optimized_Access := 'TRUE' }
VERSION : 0.1
BEGIN
END_FUNCTION

FUNCTION "STATUS RECIPE" : Void   // FC14, LAD
{ S7_Optimized_Access := 'TRUE' }
VERSION : 0.1
BEGIN
END_FUNCTION

FUNCTION "SELECT RECIPE" : Void   // FC15, LAD
{ S7_Optimized_Access := 'TRUE' }
VERSION : 0.1
BEGIN
END_FUNCTION

FUNCTION "SAVING EDIT RECIPE" : Void   // FC16, LAD
{ S7_Optimized_Access := 'TRUE' }
VERSION : 0.1
BEGIN
END_FUNCTION

FUNCTION "EDITE RECUPE ID" : Void   // FC17, LAD
{ S7_Optimized_Access := 'TRUE' }
VERSION : 0.1
BEGIN
END_FUNCTION

// folder: SAFETY

FUNCTION "RUN MODE OFF" : Void   // FC7, LAD
{ S7_Optimized_Access := 'TRUE' }
VERSION : 0.1
BEGIN
END_FUNCTION

FUNCTION "RUN MODE ON" : Void   // FC8, LAD
{ S7_Optimized_Access := 'TRUE' }
VERSION : 0.1
BEGIN
END_FUNCTION

FUNCTION "SAFETY DEVICES" : Void   // FC9, LAD
{ S7_Optimized_Access := 'TRUE' }
VERSION : 0.1
BEGIN
END_FUNCTION

FUNCTION "WATCHDOG" : Void   // FC10, LAD
{ S7_Optimized_Access := 'TRUE' }
VERSION : 0.1
BEGIN
END_FUNCTION

FUNCTION "GENERAL SAFETY" : Void   // FC18, LAD
{ S7_Optimized_Access := 'TRUE' }
VERSION : 0.1
BEGIN
END_FUNCTION

// folder: SEQUENCE

FUNCTION "INPUTS" : Void   // FC5, LAD
{ S7_Optimized_Access := 'TRUE' }
VERSION : 0.1
BEGIN
END_FUNCTION

FUNCTION "CLEAR SEQUENCE" : Void   // FC6, LAD
{ S7_Optimized_Access := 'TRUE' }
VERSION : 0.1
BEGIN
END_FUNCTION

FUNCTION "PERMISSIVES" : Void   // FC12, LAD
{ S7_Optimized_Access := 'TRUE' }
VERSION : 0.1
BEGIN
END_FUNCTION

FUNCTION "SEQUENCE" : Void   // FC19, LAD
{ S7_Optimized_Access := 'TRUE' }
VERSION : 0.1
BEGIN
END_FUNCTION

FUNCTION "OUTPUTS" : Void   // FC20, LAD
{ S7_Optimized_Access := 'TRUE' }
VERSION : 0.1
BEGIN
END_FUNCTION

// folder: UTILITIES OR DEVICES/FESTO

FUNCTION_BLOCK "FPC_PNU"   // FB4, SCL
TITLE = FPC_PNU
{ S7_Optimized_Access := 'TRUE' }
AUTHOR : FESTO
FAMILY : E-DRIVE
VERSION : 5.1
// PNU access via FPC protocol
   VAR_INPUT
      Execute : Bool;   // Perfrom Data exchange
      Write : Bool;   // Read or Write the Parameter
      DatatypeWR : Int;   // Lenth of the Paramter to Exchange in Byte(SFC and MTR only)
      PNU : Word;   // Number of the Parameter to Exchange
      Subindex : Byte;   // Subindex of the Parameter to Exchange
      Value : DInt;   // Value of the Parameter to Exchange
   END_VAR
   VAR_OUTPUT
      Done : Bool;   // Execution Done
      Error : Bool;   // Fault occured
      ActPNU : Word;   // Actual Number of the Parameter
      ActSubindex : Byte;   // Actual Subindex of the Parameter
      ActValue : DInt;   // Read Value of Parameter
      DatatypeRD : Int;   // Actual Length of the Parameter in Byte
      Status : "DT_FML_STATUS";   // Errordiscription
   END_VAR
   VAR_IN_OUT
      FML_REF : "DT_FML_REF";
   END_VAR
   VAR
      bInit : Bool := FALSE;
      TimeStart : Bool;
      lMemberID : Int := 0;
      tmpDevice : String[16];
      TONInst : TON_TIME;
      tmpStatus : "DT_FML_STATUS";
   END_VAR
   VAR CONSTANT
      TimeoutTime : Time := T#3S;
   END_VAR
BEGIN
   (*############################################################
      FESTO AG  Co., Esslingen
      Copyright (c) 2015. All rights reserved.    

      NAME OF FUNCTION BLOCK:         FPC_PNU
      VERSION NUMBER:                 V5.1
      COMPOSER:                       bejk


      -----------------------------------------------------
      Date        Name                Activity                                                                              
      06.08.2015  Benjamin Kilgus     created (V1.0)
      20.08.2015  Benjamin Kilgus     Timeout logic added (V1.1)
      07.09.2015  Benjamin Kilgus     error handling changed (V1.2)
      28.10.2015  Benjamin Kilgus     Timeout beim wegnehmen von Execute nicht abprüfen wegen bug im CMMP (V1.3)
      16.11.2015  Benjamin Kilgus     Zeile 36 --> #Status.Err := TRUE;
                                      Zeile 97 --> #TimeStart := FALSE;
                                      Option optimierter Baustein Zugriff entfernt (V1.4)      
      29.08.2016  Benjamin Klein      version changed (V4.1)
      19.10.2016  Benjamin Klein      Set ActValue in case of error to 0, tmpStatus Error fixed (V4.2)
      18.04.2017  Benjamin Klein      optimized access (V5.1)
      04.10.2017  Benjamin Klein      devicetype MTR_DCI and SFC_DC added
      20.11.2017  Benjamin Klein      copy the DataypeRD and DataypeWR(MTR and SFC only)
   ############################################################*)

   (* ====== initial block routine ===================================== *)
   (* ----- get MemberID for this function block ------------------------*)
   IF NOT #bInit THEN
       #FML_REF.MemberIDmax := #FML_REF.MemberIDmax + 1;
       #lMemberID := #FML_REF.MemberIDmax;
       #bInit := TRUE;
       #Status.Err := False;
       #Status.Cat := 1;
       #Status.ID := 1; // init active     
       RETURN;
   END_IF;

   (* ====== supervision of timeout ==================================== *)
   (* ----- timer to monitor a timeout of the function block ------------*)
   // Timout Timer
   #TONInst(IN := #TimeStart,
            PT := #TimeoutTime);

   IF #TONInst.Q THEN
       #Done := TRUE;
       #tmpStatus.Err := TRUE;
       #tmpStatus.Cat := 1;
       #tmpStatus.ID := DWORD_TO_DINT(16#8000_0014); // FB timeout         
   END_IF;

   (* ===== logic part ================================================= *)
   (* ----- ASSIGNMENT OF STATUS --------------------------------------- *)
   IF #FML_REF.MemberID = #lMemberID THEN
       IF #FML_REF.Done AND NOT #tmpStatus.Err THEN
           #TimeStart := False;
           #Done := True;
           #ActSubindex := #FML_REF.ActSubindex;
           #ActPNU := #FML_REF.ActPNU;
           #ActValue := #FML_REF.ParamValueRD;
           #DatatypeRD := #FML_REF.DatatypeRD;
           #tmpStatus.Err := False;
           #tmpStatus.Cat := 0;
           #tmpStatus.ID := 0; // none    
           IF #FML_REF.Err THEN
               #tmpStatus.Err := TRUE;
               #tmpStatus.Cat := 3;
               #tmpStatus.ID := #FML_REF.ParamValueRD; // FPC error
               #ActValue := 0;
           END_IF;
       END_IF;
   END_IF;

   (* ----- ASSIGNMENT OF CONTROL at rising edge of execute ----------- *)
   IF (#FML_REF.MemberID = 0) AND #Execute THEN
       #FML_REF.MemberID := #lMemberID;
       #TimeStart := TRUE;
       #tmpStatus.Err := FALSE;
       #tmpStatus.Cat := 1;
       #tmpStatus.ID := 16#0000_00002; // busy 

       #FML_REF.PNU := #PNU;
       #FML_REF.Subindex := #Subindex;
       #FML_REF.ParamValueWR := #Value;

       IF #Write THEN
           #FML_REF.DatatypeWR := INT_TO_BYTE(#DatatypeWR);
           #FML_REF.ReqID := 8; // write array dword        
       ELSE
           #FML_REF.ReqID := 6; //read array 
       END_IF;

       #tmpDevice := #FML_REF.DeviceType;
       IF #tmpDevice = 'EMCA_EC' OR #tmpDevice = 'CMMO_ST' THEN
           #FML_REF.FPCC_Modus := 1; // EFPC enhanced
       ELSE
           #FML_REF.FPCC_Modus := 0; // FPC Standard
       END_IF;

   ELSIF (#FML_REF.MemberID = #lMemberID) AND NOT #Execute THEN
       #FML_REF.ReqID := 0;
       #FML_REF.FPCC_Modus := 0;
       #FML_REF.PNU := 0;
       #FML_REF.Subindex := 0;
       #FML_REF.ParamValueWR := 0;
       #ActSubindex := 0;
       #ActPNU := 0;
       #ActValue := 0;
       //TimeStart         := TRUE;            (* BUG IN FIRMWARE CMMP_AS (V4.0.10.1501.13.61) --> Zeile in Lib derzeit nicht umsetzbar --> Problem am 14.09.2015 gemeldet (CHMM) *)
       IF NOT #FML_REF.Done THEN
           #FML_REF.FPCC_Modus := 0;
           #FML_REF.MemberID := 0;
           #Done := FALSE;
           #TimeStart := FALSE;
           #tmpStatus.Err := FALSE;
           #tmpStatus.Cat := 0;
           #tmpStatus.ID := 16#0000_00000; // none 
       END_IF;

   ELSIF (#FML_REF.MemberID <> #lMemberID) THEN
       IF #Execute THEN
           #tmpStatus.Err := FALSE;
           #tmpStatus.Cat := 1;
           #tmpStatus.ID := 16#0000_0000A; // other FB active
       ELSE
           #tmpStatus.Err := FALSE;
           #tmpStatus.Cat := 0;
           #tmpStatus.ID := 0; // none
       END_IF;
   END_IF;

   #Error := #tmpStatus.Err;
   #Status := #tmpStatus;
END_FUNCTION_BLOCK

FUNCTION_BLOCK "FHPP_MB_CLIENT"   // FB7, SCL
TITLE = FHPP MB_CLIENT
{ S7_Optimized_Access := 'TRUE' }
AUTHOR : FESTO
FAMILY : E-DRIVE
VERSION : 5.1
// SET and Get data from FHPP device using system function MB_CLIENT.
   VAR_INPUT
      EnableConnection : Bool;   // Freigabe zum Verbindungsaufbau
      DeviceType : String[16];   // CMMO-ST, EMCA-EC, CMMP-AS, CMMS-AS, CMMS-ST
      EnableFPC : Bool;   // Freigabe zur Verwendung von FPC-Daten
      EnableFHPPplusIn : DInt;   // FHPPplus configuration value (FCT)
      EnableFHPPplusOut : DInt;   // FHPPplus configuration value (FCT)
      IP_ADDR_Byte1 : Byte := 192;   // Erstes Byte der Server-IP-Adresse
      IP_ADDR_Byte2 : Byte := 168;   // Zweites Byte der Server-IP-Adresse
      IP_ADDR_Byte3 : Byte := 0;   // Drittes Byte der Server-IP-Adresse
      IP_ADDR_Byte4 : Byte := 207;   // Viertes Byte der Server-IP-Adresse
      InterfaceID : Hw_Any := 64;
      ConnectionID : Int := 1;   // unique connection ID (1..4095)
      TIMEOUT : Time := T#2S;
   END_VAR
   VAR_OUTPUT
      COM_ENABLED : Bool := FALSE;   // Kommunikation ist freigegeben
      Error : Bool;
      Status : "DT_FML_STATUS";
   END_VAR
   VAR_IN_OUT
      FML_REF : "DT_FML_REF";   // FHPP- und evtl. FPC-Daten die gesendet (OUT) bzw. empfangen (IN) werden
      Modbus_DATA_PTR : Variant;   // Benötigt Array [1..32] of Byte das auf Globalem DB liegt
   END_VAR
   VAR
      b_Init : Bool;
      single_Init_done : Bool;
      "STEP" : Int := 0;   // Schrittvariabel der Schrittkette
      local_IP_ADDR : Array[1..4] of Byte;   // lokale Server-IP-Adresse
      local_call_of_MB_CLIENT : MB_CLIENT;   // lokale Instanz von MB_CLIENT
      local_MB_CLIENT_Input : "DT_MB_CLIENT_INPUT";   // lokale Daten für den Aufruf von MB_CLIENT
      local_TCON_CONNECT : TCON_IP_v4;   // lokale Daten für den Aufruf von MB_CLIENT
      local_DATA_STREAM : Array[1..32] of Byte;
      TIMEOUT_Counter : TON_TIME;
      tmpFHPPplusSizeIn : DInt;
      tmpFHPPplusSizeOut : DInt;
      tmpFHPPplusElementSizeIn : Array[1..9] of DInt;
      tmpFHPPplusElementSizeOut : Array[1..9] of DInt;
      tmpStatus_MB_Client : "DT_FML_STATUS";
      tmpStatus : "DT_FML_STATUS";
      EnableFHPPplusOut_old : DInt;
      EnableFHPPplusIn_old : DInt;
      Trigger_Discon : F_TRIG;
      Trigger_Enable : R_TRIG;
      Discon_manual : Bool;
   END_VAR
   VAR_TEMP
      tmp_bRetVal : Bool;
      i : Int;
      iByteCount : DInt;
      tmpSize : DInt;
      FHPPplus24 : Array[1..24] of Byte;
      tmp : Array[1..9] of DInt;
      WORD_BYTE : Word;
      DWORD_BYTE : DInt;
   END_VAR
BEGIN
   (*############################################################
       FESTO AG  Co., Esslingen
       Copyright (c) 2015. All rights reserved.    

       NAME OF FUNCTION BLOCK:         FHPP_MB_CLIENT
       VERSION NUMBER:                 V5.1
       COMPOSER:                       bejk

       -----------------------------------------------------
      Date        Name                Activity                                                                              
      06.08.2015  Benjamin Kilgus     created (V1.0)
      15.09.2015  Benjamin Kilgus     errorhandling changed (V1.1)
      19.10.2015  Benjamin Kilgus     TIMEOUT default time auf 2000ms erhöht 
                                      Abfrage auf DeviceType ergänzt (V1.2)
      29.08.2016  Benjamin Klein      version changed (V4.1)
      17.01.2017  Christian Hammer    bugfix: reset variable "tmpStatus" at beginning, label "L_Error" and "L_NO_Error" unified
      05.07.2017  Benjamin Klein      optimized function block with Slice access instead of AT (V5.1)
      12.10.2017  Benjamin Klein      check the FHPP+size cyclic
      18.10.2017  Benjamin Klein      "tmpStatus" at beginning deleted, EnbaleConnection improved, hold communication if enablecom gets false,
                                      InterfaceID added to change the PLC port 
      16.11.2017  Benjamin Klein      ConnectionID default changed to 1
   ############################################################*)

   IF NOT #b_Init THEN
       #local_MB_CLIENT_Input.REQ := FALSE;
       #local_MB_CLIENT_Input.DISCONNECT := TRUE;
       #STEP := 0;
       #Discon_manual := false;

       // ### FHPP PLUS Input Data
       IF #EnableFHPPplusIn <> 0 THEN

           #tmpStatus.ID := "FHPPPLUS_MAPPING"(cfgFHPPplus := #EnableFHPPplusIn, FHPPplusElementSize => #tmpFHPPplusElementSizeIn, FHPPplusSize => #tmpFHPPplusSizeIn);
           #tmpFHPPplusSizeIn := #tmpFHPPplusSizeIn / 8;

           // FHPP+ Berechnung fehlerhaft beendet
           IF #tmpStatus.ID <> 0 THEN
               #tmpStatus.Err := TRUE;
               #tmpStatus.Cat := 1; // functionblock
               GOTO L_ERROR;
           END_IF;
       ELSE
           #tmpFHPPplusSizeIn := 0;
       END_IF;

       // ### FHPP PLUS Output Data
       IF #EnableFHPPplusOut <> 0 THEN

           #tmpStatus.ID := "FHPPPLUS_MAPPING"(cfgFHPPplus := #EnableFHPPplusOut, FHPPplusElementSize => #tmpFHPPplusElementSizeOut, FHPPplusSize => #tmpFHPPplusSizeOut);
           #tmpFHPPplusSizeOut := #tmpFHPPplusSizeOut / 8;

           // FHPP+ Berechnung fehlerhaft beendet
           IF #tmpStatus.ID <> 0 THEN
               #tmpStatus.Err := TRUE;
               #tmpStatus.Cat := 1; // functionblock
               GOTO L_ERROR;
           END_IF;
       ELSE
           #tmpFHPPplusSizeOut := 0;
       END_IF;
       #b_Init := TRUE;
   END_IF;
   // ### END INIT ###################################################################

   // FHPP+ size has changed
   IF #EnableFHPPplusOut <> #EnableFHPPplusOut_old OR #EnableFHPPplusIn <> #EnableFHPPplusIn_old THEN
       //new FHPP+ size -> Init the function block
       #b_Init := false;
   END_IF;

   #EnableFHPPplusIn_old := #EnableFHPPplusIn;
   #EnableFHPPplusOut_old := #EnableFHPPplusOut;

   // check device type
   IF #DeviceType = 'CMMO_ST' OR
       #DeviceType = 'EMCA_EC' OR
       #DeviceType = 'CMMP_AS' THEN

       #FML_REF.DeviceType := #DeviceType;
   ELSE
       #tmpStatus.Err := TRUE;
       #tmpStatus.Cat := 1; // functionblock
       #tmpStatus.ID := DWORD_TO_DINT(16#8000_001E); // device type not valid
       GOTO L_ERROR;
   END_IF;


   IF #local_call_of_MB_CLIENT.ERROR THEN
       #tmpStatus.Err := TRUE;
       #tmpStatus.Cat := 4;
       #tmpStatus.ID := #local_call_of_MB_CLIENT.STATUS;
       #STEP := 999;
   ELSIF #TIMEOUT_Counter.Q THEN
       #tmpStatus.Err := TRUE;
       #tmpStatus.Cat := 1;
       #tmpStatus.ID := DWORD_TO_DINT(16#8000_0014);
       #STEP := 999;
   END_IF;
   // Timeout Counter
   #TIMEOUT_Counter(IN := #single_Init_done,
                    PT := #TIMEOUT);

   // CALL the trigger Discon
   #Trigger_Discon(CLK := #EnableConnection);

   //Call the Enable Trigger
   #Trigger_Enable(CLK := #EnableConnection);

   // Verbindung abbauen
   IF #local_call_of_MB_CLIENT.Connected AND NOT #EnableConnection AND NOT #local_MB_CLIENT_Input.REQ THEN
       #local_MB_CLIENT_Input.DISCONNECT := TRUE;   //Verbindung wird abgebaut
       #single_Init_done := FALSE;
       //#local_MB_CLIENT_Input.REQ          := FALSE;
       #tmpStatus.Cat := 0;
       #tmpStatus.ID := 0;
       #tmpStatus.Err := FALSE;
       #Discon_manual := TRUE;
   ELSIF NOT #local_call_of_MB_CLIENT.Connected AND #local_call_of_MB_CLIENT.STATUS = 16#3 AND #Discon_manual THEN   // Verbindungsabbau durchgeführt
       #STEP := 0;
       #Discon_manual := FALSE;
   END_IF;

   // Check the connection
   IF #local_call_of_MB_CLIENT.Connected THEN
       #COM_ENABLED := TRUE;
   ELSE
       #COM_ENABLED    := FALSE;
   END_IF;

   // ### Modbus Conection Statemachine
   CASE #STEP OF
       0:
           IF #Trigger_Enable.Q AND #local_call_of_MB_CLIENT.STATUS = 16#7000 THEN // Freigabe fuer Verbindung und noch keine Verbindung
               #local_IP_ADDR[1] := #IP_ADDR_Byte1;
               #local_IP_ADDR[2] := #IP_ADDR_Byte2;
               #local_IP_ADDR[3] := #IP_ADDR_Byte3;
               #local_IP_ADDR[4] := #IP_ADDR_Byte4;
               #local_TCON_CONNECT.ID := INT_TO_WORD(#ConnectionID);  // eindeutige Verbindungs ID (1..4095)
               #single_Init_done := TRUE;
               #STEP := 10;
           ELSIF #Trigger_Enable.Q AND #local_call_of_MB_CLIENT.STATUS = 16#7004 AND #local_call_of_MB_CLIENT.Connected THEN //Freigabe fuer Verbindung und bereits eine Verbindung besteht
               #STEP := 20;
           ELSIF NOT #EnableConnection AND #local_call_of_MB_CLIENT.STATUS = 16#7000 THEN // Keine Freigabe fuer Verbindung und noch keine Verbindung
               ;// kein Auftrag
           ELSE
               ;// Was passiert in allen anderen Fällen? => eigentlich sofort Fehlerhandling
           END_IF;

       10: //=> Verbindung zu Server Aufbauen
           #local_MB_CLIENT_Input.DISCONNECT := false;
           #local_TCON_CONNECT.InterfaceId := #InterfaceID;      // HW-Kennung der lokalen PROFINET-Schnittstelle
           #local_TCON_CONNECT.ConnectionType := 11;
           #local_TCON_CONNECT.ActiveEstablished := TRUE;
           #local_TCON_CONNECT.RemoteAddress.ADDR := #local_IP_ADDR;
           #local_TCON_CONNECT.RemotePort := 502;     // fuer Modbus reservierter TCP-Port
           #local_TCON_CONNECT.LocalPort := 0;
           #local_MB_CLIENT_Input.MB_DATA_ADDR := 40001;

           IF #local_call_of_MB_CLIENT.STATUS = 16#1 THEN // Verbindung hergestellt.
               #single_Init_done := FALSE;
               #STEP := 15;
           ELSIF NOT #EnableConnection THEN
               #STEP := 0;
           END_IF;

       15:
           IF #local_call_of_MB_CLIENT.STATUS = 16#7004 THEN   // Verbindung hergestellt und ueberwacht.Keine Auftragsbearbeitung  aktiv.
               #STEP := 20;
           ELSIF NOT #EnableConnection THEN
               #STEP := 0;
           END_IF;

       20: //=> Schreiben der Daten mit Modbus Funktion 16 (0x10) => MB_MODE = 1 und MB_DATA_ADDR = 40001
           // Berechnung der Datenbreite für senden
           #tmpSize := 8 (*FHPP Standard*)+ (#tmpFHPPplusSizeOut);

           IF #EnableFPC THEN
               #tmpSize := #tmpSize + 8 (*FPC*);
           END_IF;
           #local_MB_CLIENT_Input.MB_DATA_LEN := DINT_TO_UINT(#tmpSize / 2); // Länge in Worte

           IF NOT #single_Init_done AND #local_call_of_MB_CLIENT.STATUS = 16#7004 AND NOT #Discon_manual THEN     //...warten, bis STATUS NICHT 0000
               #local_MB_CLIENT_Input.REQ := TRUE;
               #local_MB_CLIENT_Input.MB_MODE := 1;
               // Zusammenstellen des Modbus-Datenstroms und verschieben auf Globalen Speicher
               // FHPP STANDARD
               FOR #i := 1 TO 8 DO
                   #local_DATA_STREAM[#i] := #FML_REF.OutData.FHPP[#i];
               END_FOR;

               // FHPP FPC
               IF #EnableFPC THEN
                   FOR #i := 1 TO 8 DO
                       #local_DATA_STREAM[#i + 8] := #FML_REF.OutData.FPC[#i];
                   END_FOR;
               END_IF;

               // copy FHPPplus data from FML_REF
               IF #tmpFHPPplusSizeOut <> 0 THEN
                   #iByteCount := 1;
                   FOR #i := 1 TO 9 DO
                       CASE #tmpFHPPplusElementSizeOut[#i] OF
                           0:(* Element is empty *)
                               #iByteCount := #iByteCount + 1;// do nothing
                           8:(* Element is a BYTE *)
                               #FHPPplus24[#iByteCount] := DINT_TO_BYTE(#FML_REF.OutData.FHPPplus[#i]);
                               #iByteCount := #iByteCount + 1;
                           16:(* Element is a WORD *)
                               #WORD_BYTE := DINT_TO_WORD(#FML_REF.OutData.FHPPplus[#i]);
                               #FHPPplus24[#iByteCount] := #WORD_BYTE.%B1;
                               #FHPPplus24[#iByteCount + 1] := #WORD_BYTE.%B0;
                               #iByteCount := #iByteCount + 2;
                           32:(* Element is a DWORD *)
                               #DWORD_BYTE := (#FML_REF.OutData.FHPPplus[#i]);
                               #FHPPplus24[#iByteCount] := #DWORD_BYTE.%B3;
                               #FHPPplus24[#iByteCount + 1] := #DWORD_BYTE.%B2;
                               #FHPPplus24[#iByteCount + 2] := #DWORD_BYTE.%B1;
                               #FHPPplus24[#iByteCount + 3] := #DWORD_BYTE.%B0;
                               #iByteCount := #iByteCount + 4;
                           ELSE
                               #tmpStatus.Err := TRUE;
                               #tmpStatus.Cat := 1;
                               #tmpStatus.ID := DWORD_TO_DINT(16#8000_0001); // //no legal FHPP+ configuration
                               GOTO L_ERROR;
                       END_CASE;
                   END_FOR;
               END_IF;

               // FHPP PLUS
               IF #tmpFHPPplusSizeOut <> 0 THEN
                   #tmpSize := #tmpSize - #tmpFHPPplusSizeOut; // 8 wenn FPC FALSE, 16 wenn FPC TRUE
                   FOR #i := 1 TO #tmpFHPPplusSizeOut DO
                       #local_DATA_STREAM[#i + #tmpSize] := #FHPPplus24[#i];
                   END_FOR;
               END_IF;

               VariantPut(SRC := #local_DATA_STREAM,
                          DST := #Modbus_DATA_PTR);

               #single_Init_done := TRUE;
           ELSIF #local_call_of_MB_CLIENT.Active THEN
               #STEP := 25;
           END_IF;

       25:
           IF #single_Init_done AND #local_call_of_MB_CLIENT.DONE THEN         // Status(0000) => Anweisung wurde fehlerfrei ausgefuehr
               #single_Init_done := FALSE;
               #local_MB_CLIENT_Input.REQ := FALSE;
               #STEP := 40;
           END_IF;

       40: //=> Lesen von Daten mit Modbus Funktion 03 (0x03) => MB_MODE = 0 und MB_DATA_ADDR = 40001
           // Berechnung der Datenbreite für empfangen
           #tmpSize := 8 (*FHPP Standard*)+ (#tmpFHPPplusSizeIn);

           IF #EnableFPC THEN
               #tmpSize := #tmpSize + 8 (*FPC*);
           END_IF;
           #local_MB_CLIENT_Input.MB_DATA_LEN := DINT_TO_UINT(#tmpSize / 2); // Länge in Worte

           IF NOT #single_Init_done AND #local_call_of_MB_CLIENT.STATUS = 16#7004 AND NOT #Discon_manual THEN     //...warten, bis STATUS NICHT 0000
               #local_MB_CLIENT_Input.REQ := TRUE;
               #local_MB_CLIENT_Input.MB_MODE := 0;
               #single_Init_done := TRUE;
           ELSIF #local_call_of_MB_CLIENT.Active THEN
               #STEP := 45;
           END_IF;

       45: // Berechnung der Datenbreite für empfangen
           #tmpSize := 8 (*FHPP Standard*)+ (#tmpFHPPplusSizeIn);

           IF #EnableFPC THEN
               #tmpSize := #tmpSize + 8 (*FPC*);
           END_IF;
           #local_MB_CLIENT_Input.MB_DATA_LEN := DINT_TO_UINT(#tmpSize / 2); // Länge in Worte

           IF #single_Init_done AND #local_call_of_MB_CLIENT.DONE THEN        // Sttaus(0000) => Anweisung wurde fehlerfrei ausgefuehr
               // Holen der Daten vom Globalen Speicher und zerlegen des Modbus-Datenstroms
               VariantGet(SRC := #Modbus_DATA_PTR,
                          DST => #local_DATA_STREAM);

               // FHPP Standard
               FOR #i := 1 TO 8 DO
                   #FML_REF.InData.FHPP[#i] := #local_DATA_STREAM[#i]; //kopieren von FHPP daten in erste 8 Byte
               END_FOR;

               // FPC
               IF #EnableFPC THEN
                   FOR #i := 1 TO 8 DO
                       #FML_REF.InData.FPC[#i] := #local_DATA_STREAM[#i + 8];
                   END_FOR;
               END_IF;


               // FHPP PLUS
               IF #tmpFHPPplusSizeIn <> 0 THEN
                   #tmpSize := #tmpSize - #tmpFHPPplusSizeIn; // 8 wenn FPC FALSE, 16 wenn FPC TRUE
                   FOR #i := 1 TO #tmpFHPPplusSizeIn DO
                       #FHPPplus24[#i] := #local_DATA_STREAM[#i + #tmpSize];
                   END_FOR;
               END_IF;

               // ### copy data into FML_REF
               IF #tmpFHPPplusSizeIn <> 0 THEN
                   #iByteCount := 1;
                   FOR #i := 1 TO 9 DO
                       CASE #tmpFHPPplusElementSizeIn[#i] OF
                           0:(* Element is empty *)
                               #FML_REF.InData.FHPPplus[#i] := 0;
                               #iByteCount := #iByteCount + 1;
                           8:(* Element is a BYTE *)
                               #FML_REF.InData.FHPPplus[#i] := #FHPPplus24[#iByteCount];
                               #iByteCount := #iByteCount + 1;
                           16:(* Element is a WORD *)
                               #WORD_BYTE.%B1 := #FHPPplus24[#iByteCount];
                               #WORD_BYTE.%B0 := #FHPPplus24[#iByteCount + 1];
                               #FML_REF.InData.FHPPplus[#i] := #WORD_BYTE;
                               #iByteCount := #iByteCount + 2;

                           32:(* Element is a DWORD *)
                               #DWORD_BYTE.%B3 := #FHPPplus24[#iByteCount];
                               #DWORD_BYTE.%B2 := #FHPPplus24[#iByteCount + 1];
                               #DWORD_BYTE.%B1 := #FHPPplus24[#iByteCount + 2];
                               #DWORD_BYTE.%B0 := #FHPPplus24[#iByteCount + 3];
                               #FML_REF.InData.FHPPplus[#i] := #DWORD_BYTE;
                               #iByteCount := #iByteCount + 4;
                           ELSE
                               #tmpStatus.Err := TRUE;
                               #tmpStatus.Cat := 1;
                               #tmpStatus.ID := DWORD_TO_DINT(16#8000_0001); // //no legal FHPP+ configuration
                               GOTO L_ERROR;
                       END_CASE;
                   END_FOR;
               END_IF;

               #local_MB_CLIENT_Input.REQ := FALSE;
               #single_Init_done := FALSE;
               #STEP := 20;

           END_IF;

       999: //=> Error Handling
           #local_MB_CLIENT_Input.DISCONNECT := TRUE;   //Verbindung wird abgebaut
           #local_MB_CLIENT_Input.REQ := False;
           #single_Init_done := FALSE;  // Reset the Timer
           IF #Trigger_Discon.Q THEN           // Enable Connection falling edge in Error State
               #tmpStatus.Cat := 0;
               #tmpStatus.ID := 0;
               #tmpStatus.Err := FALSE;
               #STEP := 0;
               GOTO L_NO_ERROR;
           END_IF;
           GOTO L_ERROR;

   END_CASE;

   #tmp_bRetVal := NOT "FPC_MAPPING"(FML_REF := #FML_REF, Mode := FALSE);
   IF #tmp_bRetVal THEN
       #tmpStatus.Cat := 3; // FPC
       #tmpStatus.ID := 18;
       #tmpStatus.Err := TRUE;
       GOTO L_ERROR;
   ELSIF #tmpStatus.Err THEN
       GOTO L_ERROR;
   END_IF;

   #tmp_bRetVal := NOT "FPC_MAPPING"(FML_REF := #FML_REF, Mode := TRUE);
   IF #tmp_bRetVal THEN
       #tmpStatus.Cat := 3; // FPC
       #tmpStatus.ID := 18;
       #tmpStatus.Err := TRUE;
       GOTO L_ERROR;
   ELSIF #tmpStatus.Err THEN
       GOTO L_ERROR;
   END_IF;


   // ### EXIT ROUTINE ############################################################
   L_NO_ERROR: // LABEL
   ENO := TRUE;      // Set ENO-Bit to true
   #Status := #tmpStatus;
   #Error := #tmpStatus.Err;
   #local_call_of_MB_CLIENT(REQ := #local_MB_CLIENT_Input.REQ,
                            DISCONNECT := #local_MB_CLIENT_Input.DISCONNECT,
                            MB_MODE := #local_MB_CLIENT_Input.MB_MODE,
                            MB_DATA_ADDR := #local_MB_CLIENT_Input.MB_DATA_ADDR,
                            MB_DATA_LEN := #local_MB_CLIENT_Input.MB_DATA_LEN,
                            MB_DATA_PTR := #Modbus_DATA_PTR,
                            DONE => #local_MB_CLIENT_Input.Done,
                            BUSY => #local_MB_CLIENT_Input.Busy,
                            ERROR => #local_MB_CLIENT_Input.Error,
                            CONNECT := #local_TCON_CONNECT);


   RETURN;

   L_ERROR: // LABEL
   ENO := FALSE;     // Set ENO-Bit to false
   #Status := #tmpStatus;
   #Error := #tmpStatus.Err;
   #local_call_of_MB_CLIENT(REQ := #local_MB_CLIENT_Input.REQ,
                            DISCONNECT := #local_MB_CLIENT_Input.DISCONNECT,
                            MB_MODE := #local_MB_CLIENT_Input.MB_MODE,
                            MB_DATA_ADDR := #local_MB_CLIENT_Input.MB_DATA_ADDR,
                            MB_DATA_LEN := #local_MB_CLIENT_Input.MB_DATA_LEN,
                            MB_DATA_PTR := #Modbus_DATA_PTR,
                            DONE => #local_MB_CLIENT_Input.Done,
                            BUSY => #local_MB_CLIENT_Input.Busy,
                            ERROR => #local_MB_CLIENT_Input.Error,
                            CONNECT := #local_TCON_CONNECT);
END_FUNCTION_BLOCK

FUNCTION_BLOCK "FHPP_CTRL"   // FB10, SCL
TITLE = FHPP_CTRL
{ S7_Optimized_Access := 'TRUE' }
AUTHOR : FESTO
FAMILY : E-DRIVE
VERSION : 5.1
// control FHPP drive
   VAR_INPUT
      EnableDrive : Bool;   // Enable the Drive
      Stop : Bool;   // Stop active == 0 / Stop not active == 1
      Halt : Bool;   // Halt active == 0 / Halt not active == 1
      Brake : Bool;   // Release Brake
      ResetFault : Bool;   // Quit active Fault
      HMIAccessLocked : Bool;   // SPS Control == 1 / HMI Control == 0
      OPM : Int;   // Operation Mode CPOS
      StartTask : Bool;   // Starts Positioning Task
      StartHoming : Bool;   // Starts Homing Task
      JogPos : Bool;   // Jogging positive direction
      JogNeg : Bool;   // Jogging negaitive direction
      TeachActValue : Bool;   // Teach actual position to selected record number
      ClearRemPos : Bool;   // Clear remaining Position if Halt is/was active CDIR
      Relative : Bool;   // Absolute == 0 / Relative == 1
      DeactivateStrokeLimit : Bool;   // deactivate stroke limit (directmode/force-control)
      ExecuteFunction : Bool;   // execute cam disc function(TRUE = execute)
      RecordNo : Int;   // pre selection of the record number (Recordmode)
      SetFunctionNumber : Int;   // set cam disc function number
      SetFunctionGroup : Int;   // set cam disc function group
      SetValueVelocity : DInt;   // Setvalue Velocity (Directmode/Positionmode)
      SetValuePosition : DInt;   // pre selection Position (Directmode/Positioncontrol)
      SetValueForceRamp : DInt;   // actual value for force-ramp (directmode/force-control)
      SetValueForce : DInt;   // Setvalue Force (Directmode/Forcecontrol)
      SetValueRotRamp : DInt;   // Setvalue for Rotation-Speed-Ramp (Directmode/Rotation-Speed-Control)
      SetValueRotSpeed : DInt;   // Setvalue for Rotation-Speed (Directmode/Rotation-Speed-Control)
   END_VAR
   VAR_OUTPUT
      DriveEnabled : Bool;   // 0 == Disabled, 1 == Enabled
      Ready : Bool;   // Drive is Ready
      Warning : Bool;   // indicates Information to user (no Stop of axis)
      Fault : Bool;   // indicates Information to user (Stop of axis)
      SupplyVoltPresent : Bool;   // 0 == not present, 1 == present
      ControlFCT_HMI : Bool;   // 0 == Access MMI, 1 == SPS
      StateOPM : Int;   // State of Operation Mode (INT) SPOS
      HaltNotActive : Bool;   // 1 == Halt is not active
      AckStart : Bool;   // Acknowledge Start
      MC : Bool;   // Motioncomplete
      AckTeach : Bool;   // Acknowledge Teach
      DriveMoving : Bool;   // 1 == Drive is moving
      DragError : Bool;   // 1 == Drag Error active
      StandStillControl : Bool;   // 1 == Axis is outside tolerance window after MC
      HomingValid : Bool;   // Drive is referenced
      ActualRecordNo : Int;   // Actual Recordnumber (Recordmode)
      RC1 : Bool;   // Record Chain Condition 1 reached
      RCC : Bool;   // Record Chain Condition Complete
      VelocityLimitReached : Bool;
      StrokeLimitReached : Bool;
      FunctionIsActive : Bool;   // status of cam disc function
      ActualFunctionNumber : Int;   // actual cam disc function number
      ActualFunctionGroup : Int;   // actual cam disc function group
      ActualPosition : DInt;   // Actual Position (Directmode/Positioncontrol)
      ActualVelocity : DInt;   // Actual Velocity (Directmode)
      ActualForce : DInt;   // Actual Force (Directmode/Forcecontrol)
      ActualRotRamp : DInt;   // Actvalue FOR Rotation-Speed-Ramp (Directmode/Rotation-Speed-Control
      ActualRotSpeed : DInt;   // Actvalue FOR Rotation-Speed (Directmode/Rotation-Speed-Control
   END_VAR
   VAR_IN_OUT
      FML_REF : "DT_FML_REF";
   END_VAR
   VAR
      Converted_BYTE5_8_IN : DInt;
      Converted_BYTE5_8_OUT : DInt;
      OperationModeB1 : Bool;
      OperationModeB2 : Bool;
      ControlModeB1 : Bool;
      ControlModeB2 : Bool;
      ContinuousMode : Bool;
      StateOperationModeB1 : Bool;
      StateOperationModeB2 : Bool;
      StateControlModeB1 : Bool;
      StateControlModeB2 : Bool;
      StateContinuousMode : Bool;
   END_VAR
   VAR_TEMP
      tmpDevice : String[16];
   END_VAR
BEGIN
   (*############################################################
      FESTO AG  Co., Esslingen
      Copyright (c) 2015. All rights reserved.    

      NAME OF FUNCTION BLOCK:         FHPP_CTRL
      VERSION NUMBER:                 V5.1
      COMPOSER:                       bejk


      -----------------------------------------------------
      Date        Name                Activity                                                                              
      15.04.2015  Benjamin Kilgus     converted from Step7 V5.5 (V3.0)
      25.08.2015  Benjamin Kilgus     ActualVelocity, cast changed to BYTE_TO_SINT 
                                      case 5 for SetValue's adjusted to FW specific differents (V3.1)
      16.11.2015  Benjamin Kilgus     Änderungen für kompatibilität S7300/S7400 (V3.2)   
      13.04.2016  Benjamin Klein      Änderungen für FUNC Bit hinzugefügt
      01.08.2016  Benjamin Klein      SetValueForce wird auf 120% begrenzt, da die Rückmeldung nur 1 Byte Wertebereich hat.
      12.08.2016  Benjamin Klein      Datentyp ActualVelocity,ActualForce und ActualRotRamp auf INT geändert. 
      29.08.2016  Benjamin Klein      version changed (V4.1)
      21.09.2016  Benjamin Klein      bugfix Actual Force, limit in SetForce deactivated, SetFunctionNumber bugfix (V4.2)
      16.03.2016  Benjamin Klein      optimized function block with Slice access instead of AT (V5.1)
   ############################################################*)

   (*-----------------------------------------------------------
       Initial Block Routine
   ------------------------------------------------------------*)
   #tmpDevice := #FML_REF.DeviceType;

   (* Byte_3 *)
   #StrokeLimitReached := FALSE;
   #VelocityLimitReached := FALSE;
   #StateContinuousMode := FALSE;
   #StateControlModeB2 := FALSE;
   #StateControlModeB1 := FALSE;
   #ActualRecordNo := 0;

   (* Byte_4 *)
   #RC1 := FALSE;
   #RCC := FALSE;
   #VelocityLimitReached := FALSE;
   #StrokeLimitReached := FALSE;

   #ActualVelocity := 0;
   #ActualForce := 0;
   #ActualRotRamp := 0;

   (* Byte5-8 *)
   #ActualPosition := 0;
   #ActualRotSpeed := 0;

   (*-----------------------------------------------------------
       Asignment of the Input Data (Stateword)
   ------------------------------------------------------------*)
   #Converted_BYTE5_8_IN.%B3 := #FML_REF.InData.FHPP[5];
   #Converted_BYTE5_8_IN.%B2 := #FML_REF.InData.FHPP[6];
   #Converted_BYTE5_8_IN.%B1 := #FML_REF.InData.FHPP[7];
   #Converted_BYTE5_8_IN.%B0 := #FML_REF.InData.FHPP[8];


   (* Byte1 SCON *)

   #StateOperationModeB2 := #FML_REF.InData.FHPP[1].%X7;
   #StateOperationModeB1 := #FML_REF.InData.FHPP[1].%X6;
   #ControlFCT_HMI := #FML_REF.InData.FHPP[1].%X5;
   #SupplyVoltPresent := #FML_REF.InData.FHPP[1].%X4;
   #Fault := #FML_REF.InData.FHPP[1].%X3;
   #Warning := #FML_REF.InData.FHPP[1].%X2;
   #Ready := #FML_REF.InData.FHPP[1].%X1;
   #DriveEnabled := #FML_REF.InData.FHPP[1].%X0;

   (* Byte2 SPOS *)

   #HomingValid := #FML_REF.InData.FHPP[2].%X7;
   #StandStillControl := #FML_REF.InData.FHPP[2].%X6;
   #DragError := #FML_REF.InData.FHPP[2].%X5;
   #DriveMoving := #FML_REF.InData.FHPP[2].%X4;
   #AckTeach := #FML_REF.InData.FHPP[2].%X3;
   #MC := #FML_REF.InData.FHPP[2].%X2;
   #AckStart := #FML_REF.InData.FHPP[2].%X1;
   #HaltNotActive := #FML_REF.InData.FHPP[2].%X0;

   (* Byte_3 *)
   IF #StateOperationModeB1 THEN        // ===== directmode active =====
   (* SDIR *)

       IF #FML_REF.InData.FHPP[3].%X7 AND #tmpDevice = 'CMMP_AS' THEN

           IF #FML_REF.InData.FHPP[3].%X3 AND #FML_REF.InData.FHPP[3].%X4 THEN
               #ActualFunctionNumber := 3;
           ELSIF NOT #FML_REF.InData.FHPP[3].%X3 AND #FML_REF.InData.FHPP[3].%X4 THEN
               #ActualFunctionNumber := 2;
           ELSIF #FML_REF.InData.FHPP[3].%X3 AND NOT #FML_REF.InData.FHPP[3].%X4 THEN
               #ActualFunctionNumber := 1;
           ELSE
               #ActualFunctionNumber := 0;
           END_IF;

           IF #FML_REF.InData.FHPP[3].%X5 AND #FML_REF.InData.FHPP[3].%X6 THEN
               #ActualFunctionGroup := 3;
           ELSIF NOT #FML_REF.InData.FHPP[3].%X5 AND #FML_REF.InData.FHPP[3].%X6 THEN
               #ActualFunctionGroup := 2;
           ELSIF #FML_REF.InData.FHPP[3].%X5 AND NOT #FML_REF.InData.FHPP[3].%X6 THEN
               #ActualFunctionGroup := 1;
           ELSE
               #ActualFunctionGroup := 0;
           END_IF;

           #FunctionIsActive := TRUE;
           #StateControlModeB2 := #FML_REF.InData.FHPP[3].%X2;
           #StateControlModeB1 := #FML_REF.InData.FHPP[3].%X1;
           ;
       ELSE
           #StrokeLimitReached := #FML_REF.InData.FHPP[3].%X5;
           #VelocityLimitReached := #FML_REF.InData.FHPP[3].%X4;
           #StateContinuousMode := #FML_REF.InData.FHPP[3].%X3;
           #StateControlModeB2 := #FML_REF.InData.FHPP[3].%X2;
           #StateControlModeB1 := #FML_REF.InData.FHPP[3].%X1;

           #FunctionIsActive := FALSE;
           #ActualFunctionNumber := 0;
           #ActualFunctionGroup := 0;
       END_IF;
   ELSE                                // ===== recordmode active =====
   (* RecordNo *)
       #ActualRecordNo := BYTE_TO_INT(#FML_REF.InData.FHPP[3]);

       #FunctionIsActive := FALSE;
       #ActualFunctionNumber := 0;
       #ActualFunctionGroup := 0;
       ;
   END_IF;

   (* Coding of the Operation Mode State *)
   #StateOPM := 0;
   #StateOPM.%X0 := #StateOperationModeB1;
   #StateOPM.%X1 := #StateOperationModeB2;
   #StateOPM.%X2 := #StateControlModeB1;
   #StateOPM.%X3 := #StateControlModeB2;
   #StateOPM.%X4 := #StateContinuousMode;


   (* Byte_4/ Byte5-8*)
   CASE #StateOPM OF
       0:// (0)  Recordmode
           (* RSB record state *)

           #RC1 := #FML_REF.InData.FHPP[4].%X0;
           #RCC := #FML_REF.InData.FHPP[4].%X1;
           #VelocityLimitReached := #FML_REF.InData.FHPP[4].%X4;
           #StrokeLimitReached := #FML_REF.InData.FHPP[4].%X5;
           #ActualPosition := #Converted_BYTE5_8_IN;

       1:
           // (1)  Directmode Position Control
           #ActualVelocity := SINT_TO_DINT(#FML_REF.InData.FHPP[4]);
           #ActualPosition := #Converted_BYTE5_8_IN;

       5:// Directmode Force Control 

           #ActualForce := SINT_TO_DINT(#FML_REF.InData.FHPP[4]);
           #ActualPosition := #Converted_BYTE5_8_IN;

       9:// Directmode Rotation-Speed-Control
           #ActualRotRamp := SINT_TO_DINT(#FML_REF.InData.FHPP[4]);
           #ActualRotSpeed := #Converted_BYTE5_8_IN;
       ELSE
           ;
   END_CASE;

   (*-----------------------------------------------------------
       Asignment of the Output Data (Controlword)
   ------------------------------------------------------------*)
   (* Decoding of the Operationmode *)
   //#_Word := INT_TO_WORD(#OPM);
   #OperationModeB1 := #OPM.%X0;
   #OperationModeB2 := #OPM.%X1;
   #ControlModeB1 := #OPM.%X2;
   #ControlModeB2 := #OPM.%X3;
   #ContinuousMode := #OPM.%X4;


   (* CCON Byte_1 *)
   #FML_REF.OutData.FHPP[1].%X7 := #OperationModeB2;
   #FML_REF.OutData.FHPP[1].%X6 := #OperationModeB1; // selection of Operation Mode
   #FML_REF.OutData.FHPP[1].%X5 := #HMIAccessLocked; // get control sovereignty
   #FML_REF.OutData.FHPP[1].%X4 := false;
   #FML_REF.OutData.FHPP[1].%X3 := #ResetFault;
   #FML_REF.OutData.FHPP[1].%X2 := #Brake;
   #FML_REF.OutData.FHPP[1].%X1 := #Stop;
   #FML_REF.OutData.FHPP[1].%X0 := #EnableDrive;


   (* CPOS Byte_2 *)
   #FML_REF.OutData.FHPP[2].%X7 := FALSE;
   #FML_REF.OutData.FHPP[2].%X6 := #ClearRemPos;
   #FML_REF.OutData.FHPP[2].%X5 := #TeachActValue;
   #FML_REF.OutData.FHPP[2].%X4 := #JogNeg;
   #FML_REF.OutData.FHPP[2].%X3 := #JogPos;
   #FML_REF.OutData.FHPP[2].%X2 := #StartHoming;
   #FML_REF.OutData.FHPP[2].%X1 := #StartTask;
   #FML_REF.OutData.FHPP[2].%X0 := #Halt;

   (* Byte_3 *)
   IF #OperationModeB1 THEN     // ===== directmode =====
   (* CDIR *)
       IF #ExecuteFunction AND #tmpDevice = 'CMMP_AS' THEN
           #FML_REF.OutData.FHPP[3].%X7 := TRUE;                                          // CDIR_B7:FUNC
           #FML_REF.OutData.FHPP[3].%X6 := false;                                     // Func Group actually not used
           #FML_REF.OutData.FHPP[3].%X5 := false;                                     // Func Group actually not used
           IF #SetFunctionNumber = 3 THEN
               #FML_REF.OutData.FHPP[3].%X4 := TRUE;
               #FML_REF.OutData.FHPP[3].%X3 := TRUE;
           ELSIF #SetFunctionNumber = 2 THEN
               #FML_REF.OutData.FHPP[3].%X4 := TRUE;
               #FML_REF.OutData.FHPP[3].%X3 := FALSE;
           ELSIF #SetFunctionNumber = 1 THEN
               #FML_REF.OutData.FHPP[3].%X4 := FALSE;
               #FML_REF.OutData.FHPP[3].%X3 := TRUE;
           ELSE
               #FML_REF.OutData.FHPP[3].%X4 := FALSE;
               #FML_REF.OutData.FHPP[3].%X3 := false;
           END_IF;
           #FML_REF.OutData.FHPP[3].%X2 := #ControlModeB2;
           #FML_REF.OutData.FHPP[3].%X1 := #ControlModeB1;
           #FML_REF.OutData.FHPP[3].%X0 := #Relative;

       ELSE
           #FML_REF.OutData.FHPP[3].%X7 := FALSE;
           #FML_REF.OutData.FHPP[3].%X6 := FALSE;
           #FML_REF.OutData.FHPP[3].%X5 := #DeactivateStrokeLimit;
           #FML_REF.OutData.FHPP[3].%X4 := FALSE;
           #FML_REF.OutData.FHPP[3].%X3 := FALSE;
           #FML_REF.OutData.FHPP[3].%X2 := #ControlModeB2;
           #FML_REF.OutData.FHPP[3].%X1 := #ControlModeB1;
           #FML_REF.OutData.FHPP[3].%X0 := #Relative;
       END_IF;
   ELSE                        // ===== recordmode =====
   (* RecordNo *)
       #FML_REF.OutData.FHPP[3] := INT_TO_BYTE(#RecordNo);
   END_IF;

   (* Byte4/ Byte5-8 *)
   CASE #OPM OF
       0:// (0)  Recordmode
           #FML_REF.OutData.FHPP[4] := 0;
           #Converted_BYTE5_8_OUT := 0;

       1:
           // (1)  Directmode Position Control
           #FML_REF.OutData.FHPP[4] := DINT_TO_BYTE(MIN(IN1 := #SetValueVelocity, IN2 := 100));                   // byte 4 (permissible range of value is 0 to 100)
           #Converted_BYTE5_8_OUT := #SetValuePosition;

       5:// Directmode Forcecontrol
           (* CMMP-AS *)
           IF (#tmpDevice = 'CMMP_AS') THEN
               #FML_REF.OutData.FHPP[4] := DINT_TO_BYTE(MIN(IN1 := #SetValueForceRamp, IN2 := 100));          // byte 4 (permissible range of value is 0 to 100);
               (* CMMO-ST AND EMCA-EC *)
           ELSIF (#tmpDevice = 'CMMO_ST') OR (#tmpDevice = 'EMCA_EC') THEN
               #FML_REF.OutData.FHPP[4] := DINT_TO_BYTE(MIN(IN1 := #SetValueVelocity, IN2 := 100));
               (*other*)
           ELSE
               #FML_REF.OutData.FHPP[4] := 0;
           END_IF;

           #Converted_BYTE5_8_OUT := #SetValueForce;


       9:// Directmode Rotation-Speed-Control      
           #FML_REF.OutData.FHPP[4] := DINT_TO_BYTE(MIN(IN1 := #SetValueRotRamp, IN2 := 100));                     // byte 4 (permissible range of value is 0 to 100)
           #Converted_BYTE5_8_OUT := #SetValueRotSpeed;

       ELSE // illegal OPM              
           #FML_REF.OutData.FHPP[4] := 0;
           #Converted_BYTE5_8_OUT := 0;
   END_CASE;

   (* Set Output DATA OF DRIVE *)
   #FML_REF.OutData.FHPP[5] := #Converted_BYTE5_8_OUT.%B3;
   #FML_REF.OutData.FHPP[6] := #Converted_BYTE5_8_OUT.%B2;
   #FML_REF.OutData.FHPP[7] := #Converted_BYTE5_8_OUT.%B1;
   #FML_REF.OutData.FHPP[8] := #Converted_BYTE5_8_OUT.%B0;
END_FUNCTION_BLOCK

FUNCTION "FHPPPLUS_MAPPING" : DInt   // FC36, SCL
TITLE = FHPPPLUS_MAPPING
{ S7_Optimized_Access := 'TRUE' }
AUTHOR : FESTO
FAMILY : E-DRIVES
VERSION : 5.1
// data mapping for FHPPplus data
   VAR_INPUT
      cfgFHPPplus : DInt;
   END_VAR
   VAR_OUTPUT
      FHPPplusElementSize : Array[1..9] of DInt;
      FHPPplusSize : DInt;
   END_VAR
   VAR_TEMP
      i : Int;
      n : Int;
      tmpTeiler : DInt;
      tmpCfgFHPPplus : DInt;
      tmpElementSize : DInt;
      tmpFHPPplusSize : DInt;
   END_VAR
   VAR CONSTANT
      constTeiler : DInt := 100_000_000;
   END_VAR
BEGIN
   (*############################################################
      FESTO AG  Co., Esslingen
      Copyright (c) 2015. All rights reserved.    

      NAME OF FUNCTION BLOCK:         FHPPPLUS_MAPPING
      VERSION NUMBER:                 V5.1
      COMPOSER:                       bejk


      -----------------------------------------------------
      Date        Name                Activity                                                                              
      06.08.2015  Benjamin Kilgus     created (V1.0)
      29.08.2016  Benjamin Klein      version changed (V4.1)
      05.07.2017  Benjamin Klein      changed to optimized access (V5.1)

   ############################################################*)

   #tmpTeiler := #constTeiler;
   #tmpCfgFHPPplus := #cfgFHPPplus;
   #tmpFHPPplusSize := 0;
   #n := 1;

   // configuration 0 is not legal
   IF #cfgFHPPplus = 0 THEN
       #FHPPPLUS_MAPPING := DWORD_TO_DINT(16#8000_0001);
       RETURN;
   END_IF;

   FOR #i := 1 TO 9 DO
       #tmpElementSize := #tmpCfgFHPPplus / #tmpTeiler;
       IF #tmpElementSize = 1 OR #tmpElementSize = 2 OR #tmpElementSize = 4 THEN
           #FHPPplusElementSize[#n] := #tmpElementSize * 8; // Byte *8 = Bit
           #tmpFHPPplusSize := #tmpFHPPplusSize + #FHPPplusElementSize[#n];
           #tmpCfgFHPPplus := #tmpCfgFHPPplus - (#tmpElementSize * #tmpTeiler);
           #n := #n + 1;
       ELSIF #tmpElementSize = 0 AND #n = 1 THEN // digit empty
           #FHPPplusElementSize[10 - #i] := 0;
       ELSE
           #FHPPPLUS_MAPPING := DWORD_TO_DINT(16#8000_0001); // wrong configuration
           RETURN;
       END_IF;
       #tmpTeiler := #tmpTeiler / 10;
   END_FOR;

   IF #tmpFHPPplusSize = 64 OR #tmpFHPPplusSize = 128 OR #tmpFHPPplusSize = 192 THEN
       ;// o.k.

   ELSE // wrong size
       #FHPPPLUS_MAPPING := DWORD_TO_DINT(16#8000_0001); // function is called without legal FHPP+ configuration
       RETURN;
   END_IF;

   #FHPPplusSize := #tmpFHPPplusSize;
   #FHPPPLUS_MAPPING := 0; // o.k.
END_FUNCTION

FUNCTION "FPC_MAPPING" : Bool   // FC37, SCL
{ S7_Optimized_Access := 'TRUE' }
AUTHOR : FESTO
FAMILY : E-DRIVE
VERSION : 5.3
   VAR_INPUT
      Mode : Bool;
   END_VAR
   VAR_IN_OUT
      FML_REF : "DT_FML_REF";
   END_VAR
   VAR_TEMP
      _Word : Word;
      _DINT : DInt;
      Req_Identifier : Int;
      Resp_Identifier : Int;
   END_VAR
   VAR CONSTANT
      Const_1 : Byte := 1;
      Const_4 : Byte := 4;
   END_VAR
BEGIN
   (*############################################################
      FESTO AG  Co., Esslingen
      Copyright (c) 2015. All rights reserved.    

      NAME OF FUNCTION BLOCK:         FPC_MAPPING
      VERSION NUMBER:                 V5.3
      COMPOSER:                       bejk

   -----------------------------------------------------
      Date        Name                Activity                                                                              
      06.08.2015  Benjamin Kilgus     created (V1.0)
      07.07.2017  Benjamin Klein      version changed (V5.1)
      17.11.2017  Benjamin Klein      resp_identifier enhanced for SFC and MTR
      15.08.2019  Christian Hammer    changed to optimized block access (version 5.2)
      14.11.2019  Benjamin Klein      Bugfix of ParamValueRD=0 (version 5.3)
   ############################################################*)

   (* MAP INPUTS *)
   IF NOT #Mode THEN

       // Byte1 FPCS            
       #FML_REF.FPCS_Modus := SHR(IN := (#FML_REF.InData.FPC[1] AND 2#11110000), N := 4);

       // decoding of EFPC modus
       CASE BYTE_TO_INT(#FML_REF.FPCS_Modus) OF
           0: (* old style *)
               (* 
               -------------- Byte 1 --------------- Byte 2 ---------------------- Byte 3/4 ------------------- Byte 5..8 ----
               |  8  7  6  5  4  |  3  2  1  0  |              | 15 14 13 12 |  11  | 10 9 8 7 6 5 4 3 2 1 0 |               |
               |    FPCS Modus   |     res      |   Subindex   |      AK     |  SPM |        PNU             |     Value     |
               ---------------------------------------------------------------------------------------------------------------     
               AK:  Response Identifier (Antwortkennung)
               SPM: NOT used
               PNU: Parameternummer / Parameter-Number 
               *)
               // Byte1
               // zero in this CASE
               // Byte2  
               #FML_REF.ActSubindex := #FML_REF.InData.FPC[2];

               // Byte3/4
               #_Word.%B1 := #FML_REF.InData.FPC[3];
               #_Word.%B0 := #FML_REF.InData.FPC[4];
               #Resp_Identifier := WORD_TO_INT(SHR(IN := (#_Word AND 2#1111000000000000), N := 12));
               #FML_REF.ActPNU := #_Word AND 2#0000011111111111;

               // Byte 5..8 parameter value
               #_DINT.%B3 := #FML_REF.InData.FPC[5];
               #_DINT.%B2 := #FML_REF.InData.FPC[6];
               #_DINT.%B1 := #FML_REF.InData.FPC[7];
               #_DINT.%B0 := #FML_REF.InData.FPC[8];


           1, 2, 3:(* modus: 1 = PNU extended; 2 = KO; 3 = CAN Objects *)
               (* 
               -------------- Byte 1 --------------- Byte 2 ------------------- Byte 3/4----------------- Byte 5..8 ----
               |   7  6  5  4  |  3  2  1  0  |              | 15 14 13 12 11 10 9 8 7 6 5 4 3 2 1 0 |               |
               |  FPCS Modus   |     AK       |   Subindex   |   PNU extended or KO or CAN Object    |     Value     |
               -------------------------------------------------------------------------------------------------------       
               AK:  Response Identifier (Antwortkennung)
               *)

               // Byte 1 FPCS
               #Resp_Identifier := WORD_TO_INT(#FML_REF.InData.FPC[1] AND 2#00001111);

               // Byte 2 Subindex
               #FML_REF.ActSubindex := #FML_REF.InData.FPC[2];

               // Byte 3+4 **PKE/ PNU/ KO/ CAN**
               #FML_REF.ActPNU.%B1 := #FML_REF.InData.FPC[3];
               #FML_REF.ActPNU.%B0 := #FML_REF.InData.FPC[4];


               // Byte 5..8 parameter value
               #_DINT.%B3 := #FML_REF.InData.FPC[5];
               #_DINT.%B2 := #FML_REF.InData.FPC[6];
               #_DINT.%B1 := #FML_REF.InData.FPC[7];
               #_DINT.%B0 := #FML_REF.InData.FPC[8];


           4, 5:(* FPCS_Modus 4=Parameter File; 5=Firmware File *)
               (*
               ------ BYTE 1 ------------|-- BYTE 2 -|--BYTE 3..8 ---|
               | 7  6  5  4 | 3  2  1  0 |           |               |
               | FPCS Modus |   res      | Packet-ID |  6 BYTE Data  |
               -------------------------------------------------------        
                 Packet-ID: -------------- BYTE 2 ----------
                            | 7    6    5  | 4  3  2  1  0 |
                            | Control Bits |   Sequence-Nr |
                            -------------------------------- 
               *)
               // Byte 1 FPCS
               #Resp_Identifier := WORD_TO_INT(#FML_REF.InData.FPC[1] AND 2#00001111);
               #FML_REF.RespID := #Resp_Identifier;

               //---- Byte 2 Packet-ID ----    
               #FML_REF.FPCS_Packet.BitSequenceNr := WORD_TO_INT(#FML_REF.InData.FPC[2] AND 2#00011111);
               #FML_REF.FPCS_Packet.Control := WORD_TO_INT(SHR(IN := (#FML_REF.InData.FPC[2] AND 2#11100000), N := 5));
               //---- Byte 3..8 Data ----
               #FML_REF.FPCS_Packet.Data[1] := #FML_REF.InData.FPC[3];
               #FML_REF.FPCS_Packet.Data[2] := #FML_REF.InData.FPC[4];
               #FML_REF.FPCS_Packet.Data[3] := #FML_REF.InData.FPC[5];
               #FML_REF.FPCS_Packet.Data[4] := #FML_REF.InData.FPC[6];
               #FML_REF.FPCS_Packet.Data[5] := #FML_REF.InData.FPC[7];
               #FML_REF.FPCS_Packet.Data[6] := #FML_REF.InData.FPC[8];


           ELSE (* not implemented *)
               #FPC_MAPPING := FALSE; (* Execution was not correct *)
               RETURN;
       END_CASE;

       CASE #Resp_Identifier OF
           0, 3:(* No Transmission or Active*)
               #FML_REF.Done := FALSE;
               #FML_REF.Err := FALSE;
               #FML_REF.ActPNU := 0;
               #FML_REF.ActSubindex := 0;
               #FML_REF.ParamValueRD := 0;
               #FML_REF.DatatypeRD := 0;


           1, 4:(* Word Parameter transmittead*)
               #FML_REF.Done := TRUE;
               #FML_REF.Err := FALSE;
               #FML_REF.ParamValueRD := #_DINT;
               #FML_REF.DatatypeRD := 2;

           2, 5: (*DWord Parameter transmitted*)
               #FML_REF.Done := true;
               #FML_REF.Err := FALSE;
               #FML_REF.ParamValueRD := #_DINT;
               #FML_REF.DatatypeRD := 4;

           7:(* Transmission Failed*)
               #FML_REF.Done := TRUE;
               #FML_REF.Err := TRUE;
               #FML_REF.DatatypeRD := 0;
               #FML_REF.ParamValueRD := 0;
               #FML_REF.ActPNU := 0;


           11, 12: (*BYTE Parameter transmitted*)
               #FML_REF.Done := TRUE;
               #FML_REF.Err := False;
               #FML_REF.DatatypeRD := 1;
               #FML_REF.ParamValueRD := #_DINT;

           ELSE (* not specified*)
               #FML_REF.Done := false;
               #FML_REF.Err := TRUE;
               #FML_REF.ParamValueRD := 0;
       END_CASE;

       #FPC_MAPPING := TRUE; (* Execution was correct *)
       RETURN;

   (* MAP OUTPUTS *)
   ELSE

       IF #FML_REF.DeviceType = 'SFC_DC' OR #FML_REF.DeviceType = 'MTR_DCI' THEN
           IF #FML_REF.ReqID = 8 THEN // write
               IF BYTE_TO_INT(#FML_REF.Subindex) > 0 THEN
                   CASE BYTE_TO_INT(#FML_REF.DatatypeWR) OF
                       1:
                           #FML_REF.ReqID := 12;     //Array-Byte
                       2:
                           #FML_REF.ReqID := 7;      //Array-Wort
                       4:
                           #FML_REF.ReqID := 8;      //Array-Doppelwort
                       ELSE
                           #FPC_MAPPING := FALSE; (* wrong data type*)
                           RETURN;
                   END_CASE;
               END_IF;
               (*WRITE SINGLE PARAMETER*)
               IF #FML_REF.Subindex = 0 THEN
                   CASE BYTE_TO_INT(#FML_REF.DatatypeWR) OF
                       1:
                           #FML_REF.ReqID := 11;       // Single-Byte
                       2:
                           #FML_REF.ReqID := 2;        // Single-Wort
                       4:
                           #FML_REF.ReqID := 3;        // Single-Doppelwort
                       ELSE
                           #FPC_MAPPING := FALSE; (* wrong data type*)
                           RETURN;
                   END_CASE;
               END_IF;

           ELSIF #FML_REF.ReqID = 6 THEN
               (* READ ARRAY PARAMETER *)
               IF BYTE_TO_INT(#FML_REF.Subindex) > 0 THEN
                   #FML_REF.ReqID := 6;
               END_IF;
               (* READ SINGLE PARAMETER *)
               IF #FML_REF.Subindex = 0 THEN
                   #FML_REF.ReqID := 1;
               END_IF;
           ELSE
               ;// not specified
           END_IF;
       END_IF;
       (* create request identifier *)
       #Req_Identifier := #FML_REF.ReqID;

       CASE BYTE_TO_INT(#FML_REF.FPCC_Modus) OF
           0: (* old style *)
               (* 
               -------------- Byte 1 --------------- Byte 2 ---------------------- Byte 3 --------------------- Byte 5..8 ----
               |  8  7  6  5  4  |  3  2  1  0  |              | 15 14 13 12 |  11  | 10 9 8 7 6 5 4 3 2 1 0 |               |
               |    FPCS Modus   |     res      |   Subindex   |      AK     |  SPM |        PNU             |     Value     |
               ---------------------------------------------------------------------------------------------------------------     
               AK:  Request Identifier (Auftragskennung)
               SPM: NOT used
               PNU: Parameternummer / Parameter-Number 
               *)
               (* Byte 1 *)
               #FML_REF.OutData.FPC[1] := SHL(IN := #FML_REF.FPCC_Modus, N := 4);
               (* Byte 2 Subindex *)
               #FML_REF.OutData.FPC[2] := #FML_REF.Subindex;
               (* Byte 3+4 *)
               #_Word := SHL(IN := INT_TO_WORD(#Req_Identifier), N := 12) OR (#FML_REF.PNU AND 16#07_FF);
               #FML_REF.OutData.FPC[3] := #_Word.%B1; //Convert PKE to Byte
               #FML_REF.OutData.FPC[4] := #_Word.%B0;
               (* Byte 5..8 *)
               (* Set Output DATA OF DRIVE *)
               #FML_REF.OutData.FPC[5] := #FML_REF.ParamValueWR.%B3; //Convert PWE to Byte
               #FML_REF.OutData.FPC[6] := #FML_REF.ParamValueWR.%B2;
               #FML_REF.OutData.FPC[7] := #FML_REF.ParamValueWR.%B1;
               #FML_REF.OutData.FPC[8] := #FML_REF.ParamValueWR.%B0;

           1, 2, 3:(* modus: 1 = PNU extended; 2 = KO; 3 = CAN Objects *)
               (* 
               -------------- Byte 1 --------------- Byte 2 ------------------- Byte 3 ------------------ Byte 5..8 ----
               |  8  7  6  5  4  |  3  2  1  0  |              | 15 14 13 12 11 10 9 8 7 6 5 4 3 2 1 0 |               |
               |    FPCS Modus   |     AK       |   Subindex   |   PNU extended or KO or CAN Object    |     Value     |
               ---------------------------------------------------------------------------------------------------------       
               AK:  Request Identifier (Auftragskennung)
               *)
               (* Byte 1 *)
               #FML_REF.OutData.FPC[1] := WORD_TO_BYTE(SHL(IN := #FML_REF.FPCC_Modus, N := 4) OR INT_TO_WORD(#Req_Identifier));
               (* Byte 2 Subindex *)
               #FML_REF.OutData.FPC[2] := #FML_REF.Subindex;
               (* Byte 3+4 *)
               #FML_REF.OutData.FPC[3] := #FML_REF.PNU.%B1; //Convert PKE to Byte
               #FML_REF.OutData.FPC[4] := #FML_REF.PNU.%B0;
               (* Byte 5..8 *)
               (* Set Output DATA OF DRIVE *)
               #FML_REF.OutData.FPC[5] := #FML_REF.ParamValueWR.%B3; //Convert PWE to Byte
               #FML_REF.OutData.FPC[6] := #FML_REF.ParamValueWR.%B2;
               #FML_REF.OutData.FPC[7] := #FML_REF.ParamValueWR.%B1;
               #FML_REF.OutData.FPC[8] := #FML_REF.ParamValueWR.%B0;

           4, 5:(* FPCC_Modus 4=parameter file; 5=firmware file     
           |---------- byte 1 --------|-- byte 2 --|-- byte 3..8 ---|
           | 7  6  5  4  | 3  2  1  0 |            |                |
           |   FPCC modus |   res      | packet-ID  |  6 byte data  |
           ---------------------------------------------------------       
           Packet-ID:  | 7    6    5  | 4  3  2  1  0  |
                       | control bits |  sequence-nr   |
                       --------------------------------- *)
                       //---- byte 1 ----
                       #FML_REF.OutData.FPC[1] := WORD_TO_BYTE(SHL(IN := #FML_REF.FPCC_Modus, N := 4) OR INT_TO_WORD(#Req_Identifier));
                       //----byte 2 packet-ID ---- 
                       #FML_REF.OutData.FPC[2] := (SHL(IN := INT_TO_BYTE(#FML_REF.FPCC_Packet.Control), N := 5) OR (INT_TO_BYTE(#FML_REF.FPCC_Packet.BitSequenceNr) AND 16#1F));
                       //---- byte 3..8 data ----
                       #FML_REF.OutData.FPC[3] := #FML_REF.FPCC_Packet.Data[1];         // byte swapping for modbus data 
                       #FML_REF.OutData.FPC[4] := #FML_REF.FPCC_Packet.Data[2];
                       #FML_REF.OutData.FPC[5] := #FML_REF.FPCC_Packet.Data[3];
                       #FML_REF.OutData.FPC[6] := #FML_REF.FPCC_Packet.Data[4];
                       #FML_REF.OutData.FPC[7] := #FML_REF.FPCC_Packet.Data[5];
                       #FML_REF.OutData.FPC[8] := #FML_REF.FPCC_Packet.Data[6];

                   ELSE (* not implemented *)
                       #FPC_MAPPING := FALSE; (* Execution was not correct *)
                       RETURN;
               END_CASE;

               #FPC_MAPPING := TRUE; (* Execution was correct *)
           END_IF;
END_FUNCTION

FUNCTION "FESTO DRIVER CONTROL" : Void   // FC38, LAD
{ S7_Optimized_Access := 'TRUE' }
VERSION : 0.1
BEGIN
END_FUNCTION

FUNCTION "FESTO SET POSITION" : Void   // FC39, LAD
{ S7_Optimized_Access := 'TRUE' }
VERSION : 0.1
BEGIN
END_FUNCTION

// folder: UTILITIES OR DEVICES/KEYENCE

FUNCTION "IV RESULTS" : Void   // FC31, LAD
{ S7_Optimized_Access := 'TRUE' }
VERSION : 0.1
BEGIN
END_FUNCTION

FUNCTION "IV CONTROL" : Void   // FC32, LAD
{ S7_Optimized_Access := 'TRUE' }
VERSION : 0.1
BEGIN
END_FUNCTION

// folder: UTILITIES OR DEVICES/MODBUS TCP LABVIEW

FUNCTION "SCREEN 2 = ACTUAL RUNNIN RECIPE" : Void   // FC21, LAD
{ S7_Optimized_Access := 'TRUE' }
VERSION : 0.1
BEGIN
END_FUNCTION

FUNCTION "SCREEN 7 = SERVO FESTO" : Void   // FC22, LAD
{ S7_Optimized_Access := 'TRUE' }
VERSION : 0.1
BEGIN
END_FUNCTION

